LIN {X -205.261,Y 204.855,Z 152.881,A -44.943,B 90.000,C 0.000} C_DIS
LIN {X -207.020,Y 203.080,Z 152.821,A -44.449,B 90.000,C 0.000} C_DIS
LIN {X -207.619,Y 202.471,Z 152.789,A -44.281,B 90.000,C 0.000} C_DIS
LIN {X -208.158,Y 201.917,Z 152.576,A -44.128,B 90.000,C 0.000} C_DIS
LIN {X -208.536,Y 201.526,Z 152.267,A -44.021,B 90.000,C 0.000} C_DIS
LIN {X -208.790,Y 201.263,Z 151.819,A -43.948,B 90.000,C 0.000} C_DIS
LIN {X -208.955,Y 201.092,Z 151.191,A -43.901,B 90.000,C 0.000} C_DIS
LIN {X -209.055,Y 200.988,Z 148.696,A -43.873,B 90.000,C 0.000} C_DIS
LIN {X -209.084,Y 200.957,Z 146.196,A -43.865,B 90.000,C 0.000} C_DIS
LIN {X -209.099,Y 200.942,Z 143.696,A -43.860,B 90.000,C 0.000} C_DIS
LIN {X -209.097,Y 200.943,Z 141.196,A -43.861,B 90.000,C 0.000} C_DIS
LIN {X -209.096,Y 200.945,Z 139.404,A -43.861,B 90.000,C 0.000} C_DIS
LIN {X -208.999,Y 201.046,Z 138.325,A -43.889,B 90.000,C 0.000} C_DIS
LIN {X -208.809,Y 201.244,Z 137.619,A -43.943,B 90.000,C 0.000} C_DIS
LIN {X -208.620,Y 201.439,Z 137.220,A -43.997,B 90.000,C 0.000} C_DIS
LIN {X -208.369,Y 201.699,Z 136.948,A -44.068,B 90.000,C 0.000} C_DIS
LIN {X -208.043,Y 202.035,Z 136.793,A -44.161,B 90.000,C 0.000} C_DIS
LIN {X -207.631,Y 202.458,Z 136.749,A -44.277,B 90.000,C 0.000} C_DIS
LIN {X -206.973,Y 203.130,Z 136.893,A -44.463,B 90.000,C 0.000} C_DIS
LIN {X -205.339,Y 204.778,Z 137.822,A -44.922,B 90.000,C 0.000} C_DIS
LIN {X -203.708,Y 206.402,Z 138.797,A -45.376,B 90.000,C 0.000} C_DIS
LIN {X -202.065,Y 208.014,Z 139.772,A -45.831,B 90.000,C 0.000} C_DIS
LIN {X -200.406,Y 209.610,Z 140.748,A -46.286,B 90.000,C 0.000} C_DIS
LIN {X -198.719,Y 211.200,Z 141.683,A -46.744,B 90.000,C 0.000} C_DIS
LIN {X -197.024,Y 212.788,Z 142.609,A -47.203,B 90.000,C 0.000} C_DIS
LIN {X -195.295,Y 214.371,Z 143.478,A -47.666,B 90.000,C 0.000} C_DIS
LIN {X -193.554,Y 215.952,Z 144.325,A -48.131,B 90.000,C 0.000} C_DIS
LIN {X -191.776,Y 217.532,Z 145.096,A -48.601,B 90.000,C 0.000} C_DIS
LIN {X -189.962,Y 219.119,Z 145.758,A -49.077,B 90.000,C 0.000} C_DIS
LIN {X -189.487,Y 219.532,Z 145.914,A -49.201,B 90.000,C 0.000} C_DIS
LIN {X -188.335,Y 220.522,Z 146.091,A -49.501,B 90.000,C 0.000} C_DIS
LIN {X -187.903,Y 220.890,Z 146.053,A -49.613,B 90.000,C 0.000} C_DIS
LIN {X -187.553,Y 221.188,Z 145.936,A -49.704,B 90.000,C 0.000} C_DIS
LIN {X -187.054,Y 221.609,Z 145.542,A -49.833,B 90.000,C 0.000} C_DIS
LIN {X -186.586,Y 222.004,Z 144.866,A -49.954,B 90.000,C 0.000} C_DIS
LIN {X -186.136,Y 222.381,Z 143.887,A -50.070,B 90.000,C 0.000} C_DIS
LIN {X -185.415,Y 222.982,Z 141.569,A -50.256,B 90.000,C 0.000} C_DIS
LIN {X -184.810,Y 223.484,Z 139.196,A -50.411,B 90.000,C 0.000} C_DIS
LIN {X -184.297,Y 223.908,Z 136.787,A -50.542,B 90.000,C 0.000} C_DIS
LIN {X -183.853,Y 224.272,Z 134.354,A -50.656,B 90.000,C 0.000} C_DIS
LIN {X -183.461,Y 224.593,Z 131.906,A -50.756,B 90.000,C 0.000} C_DIS
LIN {X -183.112,Y 224.878,Z 129.447,A -50.845,B 90.000,C 0.000} C_DIS
LIN {X -182.788,Y 225.141,Z 126.982,A -50.928,B 90.000,C 0.000} C_DIS
LIN {X -182.495,Y 225.379,Z 124.511,A -51.002,B 90.000,C 0.000} C_DIS
LIN {X -182.398,Y 225.457,Z 123.827,A -51.027,B 90.000,C 0.000} C_DIS
LIN {X -182.243,Y 225.583,Z 123.542,A -51.066,B 90.000,C 0.000} C_DIS
LIN {X -181.983,Y 225.792,Z 123.296,A -51.132,B 90.000,C 0.000} C_DIS
LIN {X -181.164,Y 226.450,Z 122.936,A -51.340,B 90.000,C 0.000} C_DIS
LIN {X -180.358,Y 227.093,Z 122.834,A -51.543,B 90.000,C 0.000} C_DIS
LIN {X -179.650,Y 227.653,Z 122.887,A -51.722,B 90.000,C 0.000} C_DIS
LIN {X -179.310,Y 227.921,Z 123.049,A -51.807,B 90.000,C 0.000} C_DIS
LIN {X -179.004,Y 228.162,Z 123.312,A -51.884,B 90.000,C 0.000} C_DIS
LIN {X -178.743,Y 228.366,Z 123.666,A -51.950,B 90.000,C 0.000} C_DIS
LIN {X -178.540,Y 228.525,Z 124.096,A -52.000,B 90.000,C 0.000} C_DIS
LIN {X -178.020,Y 228.930,Z 126.507,A -52.131,B 90.000,C 0.000} C_DIS
LIN {X -177.529,Y 229.310,Z 128.928,A -52.253,B 90.000,C 0.000} C_DIS
LIN {X -177.059,Y 229.673,Z 131.357,A -52.371,B 90.000,C 0.000} C_DIS
LIN {X -176.590,Y 230.035,Z 133.785,A -52.488,B 90.000,C 0.000} C_DIS
LIN {X -176.129,Y 230.386,Z 136.217,A -52.602,B 90.000,C 0.000} C_DIS
LIN {X -175.669,Y 230.737,Z 138.649,A -52.716,B 90.000,C 0.000} C_DIS
LIN {X -175.209,Y 231.087,Z 141.081,A -52.831,B 90.000,C 0.000} C_DIS
LIN {X -174.724,Y 231.455,Z 143.506,A -52.951,B 90.000,C 0.000} C_DIS
LIN {X -174.341,Y 231.744,Z 145.063,A -53.046,B 90.000,C 0.000} C_DIS
LIN {X -174.098,Y 231.926,Z 145.616,A -53.106,B 90.000,C 0.000} C_DIS
LIN {X -173.823,Y 232.133,Z 146.029,A -53.174,B 90.000,C 0.000} C_DIS
LIN {X -173.524,Y 232.357,Z 146.285,A -53.248,B 90.000,C 0.000} C_DIS
LIN {X -172.854,Y 232.855,Z 146.429,A -53.413,B 90.000,C 0.000} C_DIS
LIN {X -171.978,Y 233.503,Z 146.327,A -53.628,B 90.000,C 0.000} C_DIS
LIN {X -170.040,Y 234.913,Z 145.614,A -54.101,B 90.000,C 0.000} C_DIS
LIN {X -168.110,Y 236.292,Z 144.829,A -54.570,B 90.000,C 0.000} C_DIS
LIN {X -166.184,Y 237.651,Z 143.995,A -55.036,B 90.000,C 0.000} C_DIS
LIN {X -164.259,Y 238.992,Z 143.132,A -55.499,B 90.000,C 0.000} C_DIS
LIN {X -162.329,Y 240.307,Z 142.239,A -55.961,B 90.000,C 0.000} C_DIS
LIN {X -160.389,Y 241.607,Z 141.346,A -56.422,B 90.000,C 0.000} C_DIS
LIN {X -158.439,Y 242.891,Z 140.453,A -56.883,B 90.000,C 0.000} C_DIS
LIN {X -156.481,Y 244.158,Z 139.554,A -57.344,B 90.000,C 0.000} C_DIS
LIN {X -154.530,Y 245.397,Z 138.599,A -57.801,B 90.000,C 0.000} C_DIS
LIN {X -152.597,Y 246.605,Z 137.574,A -58.251,B 90.000,C 0.000} C_DIS
LIN {X -151.146,Y 247.497,Z 136.837,A -58.588,B 90.000,C 0.000} C_DIS
LIN {X -150.346,Y 247.984,Z 136.687,A -58.773,B 90.000,C 0.000} C_DIS
LIN {X -149.948,Y 248.225,Z 136.710,A -58.865,B 90.000,C 0.000} C_DIS
LIN {X -149.678,Y 248.388,Z 136.816,A -58.927,B 90.000,C 0.000} C_DIS
LIN {X -149.283,Y 248.625,Z 137.164,A -59.018,B 90.000,C 0.000} C_DIS
LIN {X -148.977,Y 248.809,Z 137.712,A -59.088,B 90.000,C 0.000} C_DIS
LIN {X -148.758,Y 248.940,Z 138.468,A -59.139,B 90.000,C 0.000} C_DIS
LIN {X -148.623,Y 249.021,Z 139.439,A -59.170,B 90.000,C 0.000} C_DIS
LIN {X -148.598,Y 249.036,Z 141.939,A -59.176,B 90.000,C 0.000} C_DIS
LIN {X -148.572,Y 249.051,Z 144.439,A -59.182,B 90.000,C 0.000} C_DIS
LIN {X -148.556,Y 249.060,Z 146.939,A -59.185,B 90.000,C 0.000} C_DIS
LIN {X -148.551,Y 249.063,Z 149.439,A -59.186,B 90.000,C 0.000} C_DIS
LIN {X -148.547,Y 249.066,Z 151.587,A -59.188,B 90.000,C 0.000} C_DIS
LIN {X -147.522,Y 247.348,Z 151.587,A -59.188,B 90.000,C 0.000} C_DIS
WAIT SEC 0.1
RET=EKI_SetBool("oxy","torchState",FALSE)
RET = EKI_Send("oxy","torchState")
LIN {X -138.302,Y 231.889,Z 151.587,A -59.188,B 90.000,C 0.000} C_DIS
LIN {X -139.103,Y 231.409,Z 160.757,A -58.989,B 90.000,C 0.000} C_DIS
LIN {X -148.377,Y 246.837,Z 160.757,A -58.989,B 90.000,C 0.000} C_DIS
LIN {X -149.407,Y 248.551,Z 160.757,A -58.989,B 90.000,C 0.000} C_DIS
WAIT SEC 1
RET=EKI_SetBool("oxy","torchState",TRUE)
RET = EKI_Send("oxy","torchState")
LIN {X -148.004,Y 249.389,Z 160.848,A -59.312,B 90.000,C 0.000} C_DIS
LIN {X -147.671,Y 249.586,Z 163.317,A -59.389,B 90.000,C 0.000} C_DIS
LIN {X -147.269,Y 249.823,Z 165.773,A -59.481,B 90.000,C 0.000} C_DIS
LIN {X -147.069,Y 249.942,Z 166.758,A -59.527,B 90.000,C 0.000} C_DIS
LIN {X -146.655,Y 250.185,Z 168.058,A -59.622,B 90.000,C 0.000} C_DIS
LIN {X -146.177,Y 250.464,Z 168.917,A -59.731,B 90.000,C 0.000} C_DIS
LIN {X -145.706,Y 250.738,Z 169.357,A -59.839,B 90.000,C 0.000} C_DIS
LIN {X -144.278,Y 251.563,Z 169.869,A -60.165,B 90.000,C 0.000} C_DIS
LIN {X -143.823,Y 251.823,Z 170.248,A -60.268,B 90.000,C 0.000} C_DIS
LIN {X -143.521,Y 251.996,Z 170.826,A -60.337,B 90.000,C 0.000} C_DIS
LIN {X -143.469,Y 252.025,Z 171.669,A -60.349,B 90.000,C 0.000} C_DIS
LIN {X -143.814,Y 251.828,Z 174.137,A -60.270,B 90.000,C 0.000} C_DIS
LIN {X -144.166,Y 251.627,Z 176.604,A -60.190,B 90.000,C 0.000} C_DIS
LIN {X -144.676,Y 251.334,Z 179.034,A -60.074,B 90.000,C 0.000} C_DIS
LIN {X -145.317,Y 250.964,Z 181.422,A -59.928,B 90.000,C 0.000} C_DIS
LIN {X -146.090,Y 250.514,Z 183.756,A -59.751,B 90.000,C 0.000} C_DIS
LIN {X -146.998,Y 249.983,Z 186.024,A -59.543,B 90.000,C 0.000} C_DIS
LIN {X -148.038,Y 249.368,Z 188.213,A -59.305,B 90.000,C 0.000} C_DIS
LIN {X -149.207,Y 248.671,Z 190.310,A -59.036,B 90.000,C 0.000} C_DIS
LIN {X -150.499,Y 247.891,Z 192.302,A -58.737,B 90.000,C 0.000} C_DIS
LIN {X -151.923,Y 247.019,Z 194.163,A -58.407,B 90.000,C 0.000} C_DIS
LIN {X -153.430,Y 246.085,Z 195.926,A -58.057,B 90.000,C 0.000} C_DIS
LIN {X -155.015,Y 245.091,Z 197.583,A -57.687,B 90.000,C 0.000} C_DIS
LIN {X -156.684,Y 244.028,Z 199.112,A -57.297,B 90.000,C 0.000} C_DIS
LIN {X -158.440,Y 242.889,Z 200.479,A -56.883,B 90.000,C 0.000} C_DIS
LIN {X -160.220,Y 241.721,Z 201.789,A -56.462,B 90.000,C 0.000} C_DIS
LIN {X -161.274,Y 241.020,Z 202.510,A -56.212,B 90.000,C 0.000} C_DIS
LIN {X -161.782,Y 240.680,Z 202.765,A -56.092,B 90.000,C 0.000} C_DIS
LIN {X -161.983,Y 240.544,Z 202.607,A -56.044,B 90.000,C 0.000} C_DIS
LIN {X -162.981,Y 239.868,Z 200.417,A -55.805,B 90.000,C 0.000} C_DIS
LIN {X -163.955,Y 239.201,Z 198.214,A -55.572,B 90.000,C 0.000} C_DIS
LIN {X -164.908,Y 238.542,Z 195.998,A -55.343,B 90.000,C 0.000} C_DIS
LIN {X -165.861,Y 237.883,Z 193.783,A -55.114,B 90.000,C 0.000} C_DIS
LIN {X -166.809,Y 237.219,Z 191.567,A -54.886,B 90.000,C 0.000} C_DIS
LIN {X -167.752,Y 236.548,Z 189.351,A -54.657,B 90.000,C 0.000} C_DIS
LIN {X -168.695,Y 235.876,Z 187.136,A -54.428,B 90.000,C 0.000} C_DIS
LIN {X -169.638,Y 235.205,Z 184.920,A -54.199,B 90.000,C 0.000} C_DIS
LIN {X -170.568,Y 234.529,Z 182.700,A -53.972,B 90.000,C 0.000} C_DIS
LIN {X -171.491,Y 233.851,Z 180.478,A -53.746,B 90.000,C 0.000} C_DIS
LIN {X -172.415,Y 233.174,Z 178.256,A -53.520,B 90.000,C 0.000} C_DIS
LIN {X -173.333,Y 232.498,Z 176.031,A -53.295,B 90.000,C 0.000} C_DIS
LIN {X -174.194,Y 231.849,Z 173.775,A -53.081,B 90.000,C 0.000} C_DIS
LIN {X -175.056,Y 231.200,Z 171.520,A -52.868,B 90.000,C 0.000} C_DIS
LIN {X -175.920,Y 230.546,Z 169.268,A -52.654,B 90.000,C 0.000} C_DIS
LIN {X -176.795,Y 229.874,Z 167.024,A -52.436,B 90.000,C 0.000} C_DIS
LIN {X -177.679,Y 229.195,Z 164.787,A -52.216,B 90.000,C 0.000} C_DIS
LIN {X -178.719,Y 228.384,Z 162.663,A -51.955,B 90.000,C 0.000} C_DIS
LIN {X -179.553,Y 227.729,Z 161.118,A -51.746,B 90.000,C 0.000} C_DIS
LIN {X -179.641,Y 227.660,Z 160.788,A -51.724,B 90.000,C 0.000} C_DIS
LIN {X -177.672,Y 229.199,Z 160.786,A -52.218,B 90.000,C 0.000} C_DIS
LIN {X -175.689,Y 230.722,Z 160.784,A -52.712,B 90.000,C 0.000} C_DIS
LIN {X -173.694,Y 232.228,Z 160.782,A -53.206,B 90.000,C 0.000} C_DIS
LIN {X -171.685,Y 233.716,Z 160.780,A -53.699,B 90.000,C 0.000} C_DIS
LIN {X -169.664,Y 235.187,Z 160.778,A -54.193,B 90.000,C 0.000} C_DIS
LIN {X -167.630,Y 236.641,Z 160.776,A -54.687,B 90.000,C 0.000} C_DIS
LIN {X -165.583,Y 238.077,Z 160.774,A -55.181,B 90.000,C 0.000} C_DIS
LIN {X -163.525,Y 239.495,Z 160.772,A -55.675,B 90.000,C 0.000} C_DIS
LIN {X -161.454,Y 240.896,Z 160.769,A -56.169,B 90.000,C 0.000} C_DIS
LIN {X -159.371,Y 242.279,Z 160.767,A -56.663,B 90.000,C 0.000} C_DIS
LIN {X -157.277,Y 243.644,Z 160.765,A -57.157,B 90.000,C 0.000} C_DIS
LIN {X -155.171,Y 244.991,Z 160.763,A -57.651,B 90.000,C 0.000} C_DIS
LIN {X -153.053,Y 246.319,Z 160.761,A -58.145,B 90.000,C 0.000} C_DIS
LIN {X -150.924,Y 247.630,Z 160.759,A -58.639,B 90.000,C 0.000} C_DIS
LIN {X -149.407,Y 248.551,Z 160.757,A -58.989,B 90.000,C 0.000} C_DIS
LIN {X -148.377,Y 246.837,Z 160.757,A -58.989,B 90.000,C 0.000} C_DIS
WAIT SEC 0.1
RET=EKI_SetBool("oxy","torchState",FALSE)
RET = EKI_Send("oxy","torchState")
LIN {X -139.103,Y 231.409,Z 160.757,A -58.989,B 90.000,C 0.000} C_DIS
LIN {X -139.074,Y 231.427,Z 126.973,A -58.997,B 90.000,C 0.000} C_DIS
LIN {X -148.346,Y 246.855,Z 126.973,A -58.997,B 90.000,C 0.000} C_DIS
LIN {X -149.376,Y 248.570,Z 126.973,A -58.997,B 90.000,C 0.000} C_DIS
WAIT SEC 1
RET=EKI_SetBool("oxy","torchState",TRUE)
RET = EKI_Send("oxy","torchState")
LIN {X -149.456,Y 248.522,Z 126.964,A -58.978,B 90.000,C 0.000} C_DIS
LIN {X -151.085,Y 247.529,Z 125.348,A -58.601,B 90.000,C 0.000} C_DIS
LIN {X -152.694,Y 246.543,Z 123.709,A -58.228,B 90.000,C 0.000} C_DIS
LIN {X -154.235,Y 245.583,Z 121.990,A -57.870,B 90.000,C 0.000} C_DIS
LIN {X -155.648,Y 244.691,Z 120.131,A -57.540,B 90.000,C 0.000} C_DIS
LIN {X -156.111,Y 244.396,Z 119.238,A -57.431,B 90.000,C 0.000} C_DIS
LIN {X -156.413,Y 244.203,Z 118.302,A -57.360,B 90.000,C 0.000} C_DIS
LIN {X -156.539,Y 244.122,Z 117.113,A -57.331,B 90.000,C 0.000} C_DIS
LIN {X -156.471,Y 244.166,Z 114.614,A -57.347,B 90.000,C 0.000} C_DIS
LIN {X -156.235,Y 244.316,Z 112.130,A -57.402,B 90.000,C 0.000} C_DIS
LIN {X -155.896,Y 244.533,Z 109.663,A -57.482,B 90.000,C 0.000} C_DIS
LIN {X -155.836,Y 244.571,Z 109.402,A -57.496,B 90.000,C 0.000} C_DIS
LIN {X -153.780,Y 245.861,Z 110.003,A -57.975,B 90.000,C 0.000} C_DIS
LIN {X -151.728,Y 247.140,Z 110.635,A -58.453,B 90.000,C 0.000} C_DIS
LIN {X -149.683,Y 248.382,Z 111.361,A -58.925,B 90.000,C 0.000} C_DIS
LIN {X -149.282,Y 248.626,Z 111.504,A -59.018,B 90.000,C 0.000} C_DIS
LIN {X -149.341,Y 248.591,Z 111.613,A -59.005,B 90.000,C 0.000} C_DIS
LIN {X -151.478,Y 247.293,Z 111.578,A -58.511,B 90.000,C 0.000} C_DIS
LIN {X -153.304,Y 246.167,Z 111.730,A -58.087,B 90.000,C 0.000} C_DIS
LIN {X -154.141,Y 245.643,Z 112.053,A -57.892,B 90.000,C 0.000} C_DIS
LIN {X -154.431,Y 245.461,Z 112.286,A -57.824,B 90.000,C 0.000} C_DIS
LIN {X -154.647,Y 245.325,Z 112.591,A -57.774,B 90.000,C 0.000} C_DIS
LIN {X -154.800,Y 245.228,Z 112.983,A -57.738,B 90.000,C 0.000} C_DIS
LIN {X -154.898,Y 245.166,Z 113.481,A -57.715,B 90.000,C 0.000} C_DIS
LIN {X -154.966,Y 245.124,Z 114.860,A -57.699,B 90.000,C 0.000} C_DIS
LIN {X -154.908,Y 245.160,Z 116.152,A -57.713,B 90.000,C 0.000} C_DIS
LIN {X -154.725,Y 245.275,Z 117.383,A -57.755,B 90.000,C 0.000} C_DIS
LIN {X -154.406,Y 245.476,Z 118.611,A -57.830,B 90.000,C 0.000} C_DIS
LIN {X -153.490,Y 246.050,Z 120.865,A -58.043,B 90.000,C 0.000} C_DIS
LIN {X -152.336,Y 246.767,Z 122.963,A -58.312,B 90.000,C 0.000} C_DIS
LIN {X -150.971,Y 247.603,Z 124.883,A -58.628,B 90.000,C 0.000} C_DIS
LIN {X -149.526,Y 248.479,Z 126.726,A -58.962,B 90.000,C 0.000} C_DIS
LIN {X -149.420,Y 248.543,Z 126.863,A -58.986,B 90.000,C 0.000} C_DIS
LIN {X -149.376,Y 248.570,Z 126.973,A -58.997,B 90.000,C 0.000} C_DIS
LIN {X -148.346,Y 246.855,Z 126.973,A -58.997,B 90.000,C 0.000} C_DIS
WAIT SEC 0.1
RET=EKI_SetBool("oxy","torchState",FALSE)
RET = EKI_Send("oxy","torchState")
LIN {X -139.074,Y 231.427,Z 126.973,A -58.997,B 90.000,C 0.000} C_DIS
LIN {X -150.307,Y 224.294,Z 111.089,A -56.173,B 90.000,C 0.000} C_DIS
LIN {X -160.328,Y 239.247,Z 111.089,A -56.173,B 90.000,C 0.000} C_DIS
LIN {X -161.441,Y 240.908,Z 111.089,A -56.173,B 90.000,C 0.000} C_DIS
WAIT SEC 1
RET=EKI_SetBool("oxy","torchState",TRUE)
RET = EKI_Send("oxy","torchState")
LIN {X -163.179,Y 239.733,Z 112.449,A -55.758,B 90.000,C 0.000} C_DIS
LIN {X -164.983,Y 238.492,Z 113.656,A -55.326,B 90.000,C 0.000} C_DIS
LIN {X -166.813,Y 237.213,Z 114.780,A -54.884,B 90.000,C 0.000} C_DIS
LIN {X -168.657,Y 235.905,Z 115.847,A -54.438,B 90.000,C 0.000} C_DIS
LIN {X -170.514,Y 234.565,Z 116.848,A -53.985,B 90.000,C 0.000} C_DIS
LIN {X -172.384,Y 233.195,Z 117.786,A -53.527,B 90.000,C 0.000} C_DIS
LIN {X -174.260,Y 231.802,Z 118.674,A -53.066,B 90.000,C 0.000} C_DIS
LIN {X -176.149,Y 230.369,Z 119.466,A -52.597,B 90.000,C 0.000} C_DIS
LIN {X -178.050,Y 228.903,Z 120.165,A -52.123,B 90.000,C 0.000} C_DIS
LIN {X -178.949,Y 228.204,Z 120.474,A -51.898,B 90.000,C 0.000} C_DIS
LIN {X -180.277,Y 227.157,Z 120.647,A -51.564,B 90.000,C 0.000} C_DIS
LIN {X -181.222,Y 226.403,Z 120.632,A -51.325,B 90.000,C 0.000} C_DIS
LIN {X -182.159,Y 225.651,Z 120.471,A -51.087,B 90.000,C 0.000} C_DIS
LIN {X -184.030,Y 224.125,Z 119.823,A -50.610,B 90.000,C 0.000} C_DIS
LIN {X -185.860,Y 222.607,Z 119.050,A -50.141,B 90.000,C 0.000} C_DIS
LIN {X -187.662,Y 221.092,Z 118.209,A -49.676,B 90.000,C 0.000} C_DIS
LIN {X -189.428,Y 219.582,Z 117.288,A -49.216,B 90.000,C 0.000} C_DIS
LIN {X -191.153,Y 218.078,Z 116.282,A -48.764,B 90.000,C 0.000} C_DIS
LIN {X -192.855,Y 216.574,Z 115.237,A -48.316,B 90.000,C 0.000} C_DIS
LIN {X -194.532,Y 215.070,Z 114.152,A -47.871,B 90.000,C 0.000} C_DIS
LIN {X -196.184,Y 213.566,Z 113.032,A -47.429,B 90.000,C 0.000} C_DIS
LIN {X -197.798,Y 212.074,Z 111.839,A -46.995,B 90.000,C 0.000} C_DIS
LIN {X -199.318,Y 210.647,Z 110.461,A -46.583,B 90.000,C 0.000} C_DIS
LIN {X -200.703,Y 209.325,Z 108.853,A -46.205,B 90.000,C 0.000} C_DIS
LIN {X -202.027,Y 208.048,Z 107.160,A -45.841,B 90.000,C 0.000} C_DIS
LIN {X -203.227,Y 206.878,Z 105.448,A -45.510,B 90.000,C 0.000} C_DIS
LIN {X -203.654,Y 206.458,Z 104.627,A -45.392,B 90.000,C 0.000} C_DIS
LIN {X -203.767,Y 206.346,Z 104.238,A -45.360,B 90.000,C 0.000} C_DIS
LIN {X -203.437,Y 206.672,Z 104.386,A -45.452,B 90.000,C 0.000} C_DIS
LIN {X -201.842,Y 208.224,Z 105.524,A -45.892,B 90.000,C 0.000} C_DIS
LIN {X -200.240,Y 209.770,Z 106.660,A -46.332,B 90.000,C 0.000} C_DIS
LIN {X -198.585,Y 211.326,Z 107.705,A -46.780,B 90.000,C 0.000} C_DIS
LIN {X -196.927,Y 212.882,Z 108.743,A -47.230,B 90.000,C 0.000} C_DIS
LIN {X -195.224,Y 214.440,Z 109.704,A -47.686,B 90.000,C 0.000} C_DIS
LIN {X -193.510,Y 215.990,Z 110.657,A -48.142,B 90.000,C 0.000} C_DIS
LIN {X -191.784,Y 217.527,Z 111.610,A -48.599,B 90.000,C 0.000} C_DIS
LIN {X -190.019,Y 219.068,Z 112.483,A -49.062,B 90.000,C 0.000} C_DIS
LIN {X -188.228,Y 220.609,Z 113.298,A -49.529,B 90.000,C 0.000} C_DIS
LIN {X -186.405,Y 222.150,Z 114.042,A -50.000,B 90.000,C 0.000} C_DIS
LIN {X -184.556,Y 223.693,Z 114.712,A -50.476,B 90.000,C 0.000} C_DIS
LIN {X -182.663,Y 225.243,Z 115.226,A -50.959,B 90.000,C 0.000} C_DIS
LIN {X -182.630,Y 225.269,Z 115.234,A -50.968,B 90.000,C 0.000} C_DIS
LIN {X -180.750,Y 226.781,Z 115.482,A -51.444,B 90.000,C 0.000} C_DIS
LIN {X -178.991,Y 228.172,Z 115.427,A -51.887,B 90.000,C 0.000} C_DIS
LIN {X -177.040,Y 229.686,Z 115.037,A -52.375,B 90.000,C 0.000} C_DIS
LIN {X -175.107,Y 231.163,Z 114.462,A -52.856,B 90.000,C 0.000} C_DIS
LIN {X -173.187,Y 232.604,Z 113.764,A -53.330,B 90.000,C 0.000} C_DIS
LIN {X -171.283,Y 234.009,Z 112.956,A -53.798,B 90.000,C 0.000} C_DIS
LIN {X -169.383,Y 235.388,Z 112.098,A -54.262,B 90.000,C 0.000} C_DIS
LIN {X -167.483,Y 236.744,Z 111.203,A -54.723,B 90.000,C 0.000} C_DIS
LIN {X -165.603,Y 238.066,Z 110.221,A -55.177,B 90.000,C 0.000} C_DIS
LIN {X -163.709,Y 239.370,Z 109.238,A -55.631,B 90.000,C 0.000} C_DIS
LIN {X -161.828,Y 240.641,Z 108.193,A -56.080,B 90.000,C 0.000} C_DIS
LIN {X -159.951,Y 241.900,Z 107.124,A -56.526,B 90.000,C 0.000} C_DIS
LIN {X -158.082,Y 243.120,Z 105.998,A -56.967,B 90.000,C 0.000} C_DIS
LIN {X -156.203,Y 244.337,Z 104.884,A -57.409,B 90.000,C 0.000} C_DIS
LIN {X -156.076,Y 244.418,Z 104.809,A -57.439,B 90.000,C 0.000} C_DIS
LIN {X -155.819,Y 244.582,Z 104.709,A -57.500,B 90.000,C 0.000} C_DIS
LIN {X -155.735,Y 244.635,Z 104.743,A -57.519,B 90.000,C 0.000} C_DIS
LIN {X -156.034,Y 244.445,Z 105.280,A -57.449,B 90.000,C 0.000} C_DIS
LIN {X -157.532,Y 243.480,Z 107.034,A -57.097,B 90.000,C 0.000} C_DIS
LIN {X -159.067,Y 242.480,Z 108.735,A -56.735,B 90.000,C 0.000} C_DIS
LIN {X -160.666,Y 241.423,Z 110.339,A -56.356,B 90.000,C 0.000} C_DIS
LIN {X -161.441,Y 240.908,Z 111.089,A -56.173,B 90.000,C 0.000} C_DIS
LIN {X -160.328,Y 239.247,Z 111.089,A -56.173,B 90.000,C 0.000} C_DIS
WAIT SEC 0.1
RET=EKI_SetBool("oxy","torchState",FALSE)
RET = EKI_Send("oxy","torchState")
LIN {X -150.307,Y 224.294,Z 111.089,A -56.173,B 90.000,C 0.000} C_DIS
LIN {X -152.164,Y 223.038,Z 106.199,A -55.697,B 90.000,C 0.000} C_DIS
LIN {X -162.308,Y 237.908,Z 106.199,A -55.697,B 90.000,C 0.000} C_DIS
LIN {X -163.435,Y 239.560,Z 106.199,A -55.697,B 90.000,C 0.000} C_DIS
WAIT SEC 1
RET=EKI_SetBool("oxy","torchState",TRUE)
RET = EKI_Send("oxy","torchState")
LIN {X -163.575,Y 239.464,Z 106.192,A -55.663,B 90.000,C 0.000} C_DIS
LIN {X -163.681,Y 239.392,Z 106.136,A -55.638,B 90.000,C 0.000} C_DIS
LIN {X -163.820,Y 239.297,Z 105.921,A -55.605,B 90.000,C 0.000} C_DIS
LIN {X -164.813,Y 238.612,Z 103.731,A -55.367,B 90.000,C 0.000} C_DIS
LIN {X -165.781,Y 237.936,Z 101.527,A -55.133,B 90.000,C 0.000} C_DIS
LIN {X -166.748,Y 237.260,Z 99.324,A -54.900,B 90.000,C 0.000} C_DIS
LIN {X -167.714,Y 236.582,Z 97.120,A -54.667,B 90.000,C 0.000} C_DIS
LIN {X -168.674,Y 235.894,Z 94.916,A -54.434,B 90.000,C 0.000} C_DIS
LIN {X -169.634,Y 235.206,Z 92.713,A -54.200,B 90.000,C 0.000} C_DIS
LIN {X -170.593,Y 234.516,Z 90.510,A -53.967,B 90.000,C 0.000} C_DIS
LIN {X -171.553,Y 233.815,Z 88.311,A -53.732,B 90.000,C 0.000} C_DIS
LIN {X -172.450,Y 233.154,Z 86.368,A -53.512,B 90.000,C 0.000} C_DIS
LIN {X -173.673,Y 232.242,Z 84.387,A -53.210,B 90.000,C 0.000} C_DIS
LIN {X -174.914,Y 231.307,Z 82.429,A -52.903,B 90.000,C 0.000} C_DIS
LIN {X -175.617,Y 230.778,Z 81.320,A -52.730,B 90.000,C 0.000} C_DIS
LIN {X -175.703,Y 230.713,Z 80.905,A -52.708,B 90.000,C 0.000} C_DIS
LIN {X -175.604,Y 230.789,Z 80.135,A -52.733,B 90.000,C 0.000} C_DIS
LIN {X -174.968,Y 231.270,Z 77.766,A -52.891,B 90.000,C 0.000} C_DIS
LIN {X -174.142,Y 231.893,Z 75.490,A -53.095,B 90.000,C 0.000} C_DIS
LIN {X -174.024,Y 231.982,Z 75.194,A -53.124,B 90.000,C 0.000} C_DIS
LIN {X -173.228,Y 232.577,Z 73.722,A -53.321,B 90.000,C 0.000} C_DIS
LIN {X -172.272,Y 233.286,Z 72.382,A -53.556,B 90.000,C 0.000} C_DIS
LIN {X -171.261,Y 234.029,Z 71.262,A -53.804,B 90.000,C 0.000} C_DIS
LIN {X -170.170,Y 234.824,Z 70.335,A -54.070,B 90.000,C 0.000} C_DIS
LIN {X -168.953,Y 235.701,Z 69.568,A -54.367,B 90.000,C 0.000} C_DIS
LIN {X -167.565,Y 236.690,Z 68.928,A -54.703,B 90.000,C 0.000} C_DIS
LIN {X -166.410,Y 237.503,Z 68.568,A -54.982,B 90.000,C 0.000} C_DIS
LIN {X -164.358,Y 238.927,Z 68.468,A -55.476,B 90.000,C 0.000} C_DIS
LIN {X -164.146,Y 239.074,Z 68.470,A -55.527,B 90.000,C 0.000} C_DIS
LIN {X -164.072,Y 239.125,Z 68.526,A -55.545,B 90.000,C 0.000} C_DIS
LIN {X -164.188,Y 239.045,Z 68.748,A -55.517,B 90.000,C 0.000} C_DIS
LIN {X -164.530,Y 238.809,Z 69.148,A -55.435,B 90.000,C 0.000} C_DIS
LIN {X -166.385,Y 237.520,Z 70.220,A -54.988,B 90.000,C 0.000} C_DIS
LIN {X -168.178,Y 236.254,Z 71.417,A -54.555,B 90.000,C 0.000} C_DIS
LIN {X -169.310,Y 235.445,Z 72.362,A -54.280,B 90.000,C 0.000} C_DIS
LIN {X -170.408,Y 234.651,Z 73.551,A -54.012,B 90.000,C 0.000} C_DIS
LIN {X -171.502,Y 233.853,Z 75.196,A -53.745,B 90.000,C 0.000} C_DIS
LIN {X -171.887,Y 233.570,Z 76.039,A -53.650,B 90.000,C 0.000} C_DIS
LIN {X -172.172,Y 233.360,Z 76.912,A -53.580,B 90.000,C 0.000} C_DIS
LIN {X -172.418,Y 233.178,Z 78.168,A -53.520,B 90.000,C 0.000} C_DIS
LIN {X -172.458,Y 233.149,Z 79.528,A -53.510,B 90.000,C 0.000} C_DIS
LIN {X -172.301,Y 233.264,Z 81.162,A -53.548,B 90.000,C 0.000} C_DIS
LIN {X -171.868,Y 233.584,Z 82.885,A -53.655,B 90.000,C 0.000} C_DIS
LIN {X -171.047,Y 234.183,Z 85.169,A -53.856,B 90.000,C 0.000} C_DIS
LIN {X -170.227,Y 234.782,Z 87.453,A -54.056,B 90.000,C 0.000} C_DIS
LIN {X -169.376,Y 235.390,Z 89.724,A -54.263,B 90.000,C 0.000} C_DIS
LIN {X -168.518,Y 236.001,Z 91.991,A -54.471,B 90.000,C 0.000} C_DIS
LIN {X -167.659,Y 236.612,Z 94.258,A -54.679,B 90.000,C 0.000} C_DIS
LIN {X -166.801,Y 237.223,Z 96.525,A -54.887,B 90.000,C 0.000} C_DIS
LIN {X -165.941,Y 237.829,Z 98.793,A -55.095,B 90.000,C 0.000} C_DIS
LIN {X -165.079,Y 238.425,Z 101.062,A -55.302,B 90.000,C 0.000} C_DIS
LIN {X -164.216,Y 239.021,Z 103.332,A -55.509,B 90.000,C 0.000} C_DIS
LIN {X -163.353,Y 239.616,Z 105.601,A -55.717,B 90.000,C 0.000} C_DIS
LIN {X -163.328,Y 239.633,Z 105.669,A -55.723,B 90.000,C 0.000} C_DIS
LIN {X -163.291,Y 239.658,Z 105.884,A -55.731,B 90.000,C 0.000} C_DIS
LIN {X -163.352,Y 239.617,Z 106.124,A -55.717,B 90.000,C 0.000} C_DIS
LIN {X -163.435,Y 239.560,Z 106.199,A -55.697,B 90.000,C 0.000} C_DIS
LIN {X -162.308,Y 237.908,Z 106.199,A -55.697,B 90.000,C 0.000} C_DIS
WAIT SEC 0.1
RET=EKI_SetBool("oxy","torchState",FALSE)
RET = EKI_Send("oxy","torchState")
LIN {X -152.164,Y 223.038,Z 106.199,A -55.697,B 90.000,C 0.000} C_DIS
LIN {X -141.870,Y 229.724,Z 103.032,A -58.302,B 90.000,C 0.000} C_DIS
LIN {X -151.328,Y 245.038,Z 103.032,A -58.302,B 90.000,C 0.000} C_DIS
LIN {X -152.379,Y 246.740,Z 103.032,A -58.302,B 90.000,C 0.000} C_DIS
WAIT SEC 1
RET=EKI_SetBool("oxy","torchState",TRUE)
RET = EKI_Send("oxy","torchState")
LIN {X -152.409,Y 246.722,Z 102.859,A -58.295,B 90.000,C 0.000} C_DIS
LIN {X -152.288,Y 246.796,Z 102.521,A -58.323,B 90.000,C 0.000} C_DIS
LIN {X -150.312,Y 248.003,Z 101.580,A -58.780,B 90.000,C 0.000} C_DIS
LIN {X -148.374,Y 249.167,Z 100.511,A -59.227,B 90.000,C 0.000} C_DIS
LIN {X -147.908,Y 249.446,Z 100.241,A -59.334,B 90.000,C 0.000} C_DIS
LIN {X -146.106,Y 250.505,Z 98.870,A -59.747,B 90.000,C 0.000} C_DIS
LIN {X -144.571,Y 251.395,Z 97.332,A -60.098,B 90.000,C 0.000} C_DIS
LIN {X -143.328,Y 252.105,Z 95.636,A -60.381,B 90.000,C 0.000} C_DIS
LIN {X -142.342,Y 252.664,Z 93.741,A -60.605,B 90.000,C 0.000} C_DIS
LIN {X -141.786,Y 252.976,Z 92.230,A -60.731,B 90.000,C 0.000} C_DIS
LIN {X -141.389,Y 253.198,Z 90.624,A -60.820,B 90.000,C 0.000} C_DIS
LIN {X -141.111,Y 253.353,Z 88.144,A -60.883,B 90.000,C 0.000} C_DIS
LIN {X -141.044,Y 253.390,Z 85.900,A -60.898,B 90.000,C 0.000} C_DIS
LIN {X -140.787,Y 253.533,Z 86.205,A -60.957,B 90.000,C 0.000} C_DIS
LIN {X -140.484,Y 253.701,Z 86.731,A -61.025,B 90.000,C 0.000} C_DIS
LIN {X -140.301,Y 253.802,Z 88.839,A -61.066,B 90.000,C 0.000} C_DIS
LIN {X -140.331,Y 253.786,Z 91.236,A -61.060,B 90.000,C 0.000} C_DIS
LIN {X -140.568,Y 253.655,Z 92.829,A -61.006,B 90.000,C 0.000} C_DIS
LIN {X -140.966,Y 253.433,Z 94.320,A -60.916,B 90.000,C 0.000} C_DIS
LIN {X -141.527,Y 253.121,Z 95.713,A -60.789,B 90.000,C 0.000} C_DIS
LIN {X -142.251,Y 252.715,Z 97.010,A -60.625,B 90.000,C 0.000} C_DIS
LIN {X -143.287,Y 252.128,Z 98.343,A -60.390,B 90.000,C 0.000} C_DIS
LIN {X -144.455,Y 251.462,Z 99.548,A -60.124,B 90.000,C 0.000} C_DIS
LIN {X -145.928,Y 250.610,Z 100.652,A -59.788,B 90.000,C 0.000} C_DIS
LIN {X -147.583,Y 249.638,Z 101.587,A -59.409,B 90.000,C 0.000} C_DIS
LIN {X -149.609,Y 248.428,Z 102.411,A -58.943,B 90.000,C 0.000} C_DIS
LIN {X -151.685,Y 247.167,Z 103.004,A -58.463,B 90.000,C 0.000} C_DIS
LIN {X -152.252,Y 246.819,Z 103.103,A -58.331,B 90.000,C 0.000} C_DIS
LIN {X -152.379,Y 246.740,Z 103.032,A -58.302,B 90.000,C 0.000} C_DIS
LIN {X -151.328,Y 245.038,Z 103.032,A -58.302,B 90.000,C 0.000} C_DIS
WAIT SEC 0.1
RET=EKI_SetBool("oxy","torchState",FALSE)
RET = EKI_Send("oxy","torchState")
LIN {X -141.870,Y 229.724,Z 103.032,A -58.302,B 90.000,C 0.000} C_DIS
LIN {X -131.390,Y 235.874,Z 104.704,A -60.881,B 90.000,C 0.000} C_DIS
LIN {X -140.149,Y 251.599,Z 104.704,A -60.881,B 90.000,C 0.000} C_DIS
LIN {X -141.123,Y 253.346,Z 104.704,A -60.881,B 90.000,C 0.000} C_DIS
WAIT SEC 1
RET=EKI_SetBool("oxy","torchState",TRUE)
RET = EKI_Send("oxy","torchState")
LIN {X -139.117,Y 254.450,Z 105.709,A -61.333,B 90.000,C 0.000} C_DIS
LIN {X -138.204,Y 254.950,Z 106.149,A -61.539,B 90.000,C 0.000} C_DIS
LIN {X -136.189,Y 256.032,Z 106.784,A -61.991,B 90.000,C 0.000} C_DIS
LIN {X -135.810,Y 256.234,Z 106.779,A -62.075,B 90.000,C 0.000} C_DIS
LIN {X -135.472,Y 256.412,Z 106.322,A -62.151,B 90.000,C 0.000} C_DIS
LIN {X -134.399,Y 256.975,Z 104.136,A -62.390,B 90.000,C 0.000} C_DIS
LIN {X -133.416,Y 257.488,Z 101.895,A -62.609,B 90.000,C 0.000} C_DIS
LIN {X -132.809,Y 257.802,Z 99.760,A -62.744,B 90.000,C 0.000} C_DIS
LIN {X -132.638,Y 257.890,Z 98.389,A -62.782,B 90.000,C 0.000} C_DIS
LIN {X -134.601,Y 256.866,Z 97.228,A -62.345,B 90.000,C 0.000} C_DIS
LIN {X -136.545,Y 255.843,Z 96.035,A -61.911,B 90.000,C 0.000} C_DIS
LIN {X -137.518,Y 255.319,Z 98.277,A -61.692,B 90.000,C 0.000} C_DIS
LIN {X -138.472,Y 254.804,Z 100.530,A -61.478,B 90.000,C 0.000} C_DIS
LIN {X -139.618,Y 254.178,Z 102.662,A -61.220,B 90.000,C 0.000} C_DIS
LIN {X -140.014,Y 253.961,Z 103.282,A -61.131,B 90.000,C 0.000} C_DIS
LIN {X -141.048,Y 253.388,Z 104.532,A -60.898,B 90.000,C 0.000} C_DIS
LIN {X -141.123,Y 253.346,Z 104.704,A -60.881,B 90.000,C 0.000} C_DIS
LIN {X -140.149,Y 251.599,Z 104.704,A -60.881,B 90.000,C 0.000} C_DIS
WAIT SEC 0.1
RET=EKI_SetBool("oxy","torchState",FALSE)
RET = EKI_Send("oxy","torchState")
LIN {X -131.390,Y 235.874,Z 104.704,A -60.881,B 90.000,C 0.000} C_DIS
LIN {X -124.578,Y 239.542,Z 107.483,A -62.522,B 90.000,C 0.000} C_DIS
LIN {X -132.883,Y 255.511,Z 107.483,A -62.522,B 90.000,C 0.000} C_DIS
LIN {X -133.806,Y 257.286,Z 107.483,A -62.522,B 90.000,C 0.000} C_DIS
WAIT SEC 1
RET=EKI_SetBool("oxy","torchState",TRUE)
RET = EKI_Send("oxy","torchState")
LIN {X -132.836,Y 257.788,Z 105.235,A -62.738,B 90.000,C 0.000} C_DIS
LIN {X -132.043,Y 258.195,Z 102.899,A -62.914,B 90.000,C 0.000} C_DIS
LIN {X -131.462,Y 258.491,Z 100.486,A -63.043,B 90.000,C 0.000} C_DIS
LIN {X -131.165,Y 258.642,Z 98.370,A -63.109,B 90.000,C 0.000} C_DIS
LIN {X -131.194,Y 258.627,Z 95.870,A -63.103,B 90.000,C 0.000} C_DIS
LIN {X -131.290,Y 258.578,Z 94.495,A -63.081,B 90.000,C 0.000} C_DIS
LIN {X -131.688,Y 258.376,Z 92.520,A -62.993,B 90.000,C 0.000} C_DIS
LIN {X -132.314,Y 258.056,Z 90.651,A -62.854,B 90.000,C 0.000} C_DIS
LIN {X -133.194,Y 257.603,Z 88.853,A -62.659,B 90.000,C 0.000} C_DIS
LIN {X -134.306,Y 257.025,Z 87.164,A -62.411,B 90.000,C 0.000} C_DIS
LIN {X -135.864,Y 256.204,Z 85.389,A -62.063,B 90.000,C 0.000} C_DIS
LIN {X -137.578,Y 255.288,Z 83.817,A -61.679,B 90.000,C 0.000} C_DIS
LIN {X -139.395,Y 254.294,Z 82.417,A -61.270,B 90.000,C 0.000} C_DIS
LIN {X -141.223,Y 253.289,Z 81.039,A -60.858,B 90.000,C 0.000} C_DIS
LIN {X -142.847,Y 252.378,Z 79.808,A -60.490,B 90.000,C 0.000} C_DIS
LIN {X -143.257,Y 252.146,Z 79.046,A -60.397,B 90.000,C 0.000} C_DIS
LIN {X -143.083,Y 252.244,Z 79.057,A -60.436,B 90.000,C 0.000} C_DIS
LIN {X -141.199,Y 253.304,Z 79.811,A -60.863,B 90.000,C 0.000} C_DIS
LIN {X -139.222,Y 254.386,Z 80.893,A -61.309,B 90.000,C 0.000} C_DIS
LIN {X -137.262,Y 255.458,Z 81.967,A -61.750,B 90.000,C 0.000} C_DIS
LIN {X -135.518,Y 256.387,Z 83.498,A -62.141,B 90.000,C 0.000} C_DIS
LIN {X -133.866,Y 257.253,Z 85.163,A -62.509,B 90.000,C 0.000} C_DIS
LIN {X -133.271,Y 257.563,Z 85.815,A -62.642,B 90.000,C 0.000} C_DIS
LIN {X -132.193,Y 258.118,Z 87.299,A -62.881,B 90.000,C 0.000} C_DIS
LIN {X -131.331,Y 258.558,Z 88.852,A -63.072,B 90.000,C 0.000} C_DIS
LIN {X -130.682,Y 258.887,Z 90.480,A -63.216,B 90.000,C 0.000} C_DIS
LIN {X -130.036,Y 259.211,Z 92.873,A -63.359,B 90.000,C 0.000} C_DIS
LIN {X -129.670,Y 259.395,Z 94.776,A -63.440,B 90.000,C 0.000} C_DIS
LIN {X -129.587,Y 259.436,Z 97.274,A -63.458,B 90.000,C 0.000} C_DIS
LIN {X -129.673,Y 259.394,Z 99.271,A -63.439,B 90.000,C 0.000} C_DIS
LIN {X -130.023,Y 259.218,Z 101.311,A -63.362,B 90.000,C 0.000} C_DIS
LIN {X -130.550,Y 258.953,Z 103.240,A -63.245,B 90.000,C 0.000} C_DIS
LIN {X -131.476,Y 258.484,Z 105.514,A -63.040,B 90.000,C 0.000} C_DIS
LIN {X -132.625,Y 257.896,Z 107.655,A -62.785,B 90.000,C 0.000} C_DIS
LIN {X -133.052,Y 257.677,Z 108.353,A -62.690,B 90.000,C 0.000} C_DIS
LIN {X -134.452,Y 256.949,Z 110.072,A -62.379,B 90.000,C 0.000} C_DIS
LIN {X -134.918,Y 256.704,Z 109.985,A -62.275,B 90.000,C 0.000} C_DIS
LIN {X -133.925,Y 257.224,Z 107.751,A -62.496,B 90.000,C 0.000} C_DIS
LIN {X -133.806,Y 257.286,Z 107.483,A -62.522,B 90.000,C 0.000} C_DIS
LIN {X -132.883,Y 255.511,Z 107.483,A -62.522,B 90.000,C 0.000} C_DIS
WAIT SEC 0.1
RET=EKI_SetBool("oxy","torchState",FALSE)
RET = EKI_Send("oxy","torchState")
LIN {X -124.578,Y 239.542,Z 107.483,A -62.522,B 90.000,C 0.000} C_DIS
LIN {X -147.605,Y 226.082,Z 82.780,A -56.860,B 90.000,C 0.000} C_DIS
LIN {X -157.445,Y 241.154,Z 82.780,A -56.860,B 90.000,C 0.000} C_DIS
LIN {X -158.538,Y 242.828,Z 82.780,A -56.860,B 90.000,C 0.000} C_DIS
WAIT SEC 1
RET=EKI_SetBool("oxy","torchState",TRUE)
RET = EKI_Send("oxy","torchState")
LIN {X -159.334,Y 242.307,Z 83.710,A -56.672,B 90.000,C 0.000} C_DIS
LIN {X -160.292,Y 241.675,Z 84.484,A -56.446,B 90.000,C 0.000} C_DIS
LIN {X -161.353,Y 240.967,Z 85.049,A -56.193,B 90.000,C 0.000} C_DIS
LIN {X -162.153,Y 240.429,Z 85.292,A -56.003,B 90.000,C 0.000} C_DIS
LIN {X -163.942,Y 239.213,Z 85.458,A -55.576,B 90.000,C 0.000} C_DIS
LIN {X -164.767,Y 238.646,Z 85.365,A -55.378,B 90.000,C 0.000} C_DIS
LIN {X -165.607,Y 238.064,Z 85.121,A -55.176,B 90.000,C 0.000} C_DIS
LIN {X -166.392,Y 237.516,Z 84.749,A -54.987,B 90.000,C 0.000} C_DIS
LIN {X -167.114,Y 237.008,Z 84.259,A -54.812,B 90.000,C 0.000} C_DIS
LIN {X -167.764,Y 236.549,Z 83.660,A -54.655,B 90.000,C 0.000} C_DIS
LIN {X -168.333,Y 236.144,Z 82.963,A -54.517,B 90.000,C 0.000} C_DIS
LIN {X -168.812,Y 235.802,Z 82.177,A -54.401,B 90.000,C 0.000} C_DIS
LIN {X -169.192,Y 235.529,Z 81.313,A -54.308,B 90.000,C 0.000} C_DIS
LIN {X -169.465,Y 235.333,Z 80.379,A -54.242,B 90.000,C 0.000} C_DIS
LIN {X -169.617,Y 235.224,Z 79.076,A -54.205,B 90.000,C 0.000} C_DIS
LIN {X -169.534,Y 235.283,Z 77.767,A -54.225,B 90.000,C 0.000} C_DIS
LIN {X -169.315,Y 235.441,Z 76.834,A -54.279,B 90.000,C 0.000} C_DIS
LIN {X -168.984,Y 235.678,Z 75.969,A -54.359,B 90.000,C 0.000} C_DIS
LIN {X -168.548,Y 235.991,Z 75.178,A -54.465,B 90.000,C 0.000} C_DIS
LIN {X -168.012,Y 236.373,Z 74.468,A -54.595,B 90.000,C 0.000} C_DIS
LIN {X -167.381,Y 236.820,Z 73.845,A -54.748,B 90.000,C 0.000} C_DIS
LIN {X -166.662,Y 237.326,Z 73.318,A -54.922,B 90.000,C 0.000} C_DIS
LIN {X -165.861,Y 237.887,Z 72.893,A -55.115,B 90.000,C 0.000} C_DIS
LIN {X -164.982,Y 238.497,Z 72.578,A -55.326,B 90.000,C 0.000} C_DIS
LIN {X -163.701,Y 239.378,Z 72.436,A -55.633,B 90.000,C 0.000} C_DIS
LIN {X -162.418,Y 240.251,Z 72.504,A -55.940,B 90.000,C 0.000} C_DIS
LIN {X -161.463,Y 240.893,Z 72.794,A -56.167,B 90.000,C 0.000} C_DIS
LIN {X -160.595,Y 241.473,Z 73.220,A -56.374,B 90.000,C 0.000} C_DIS
LIN {X -159.803,Y 241.998,Z 73.788,A -56.561,B 90.000,C 0.000} C_DIS
LIN {X -159.078,Y 242.475,Z 74.504,A -56.733,B 90.000,C 0.000} C_DIS
LIN {X -158.472,Y 242.871,Z 75.294,A -56.876,B 90.000,C 0.000} C_DIS
LIN {X -157.996,Y 243.181,Z 76.134,A -56.988,B 90.000,C 0.000} C_DIS
LIN {X -157.652,Y 243.404,Z 77.015,A -57.069,B 90.000,C 0.000} C_DIS
LIN {X -157.442,Y 243.541,Z 77.929,A -57.119,B 90.000,C 0.000} C_DIS
LIN {X -157.366,Y 243.590,Z 78.868,A -57.136,B 90.000,C 0.000} C_DIS
LIN {X -157.426,Y 243.551,Z 79.823,A -57.122,B 90.000,C 0.000} C_DIS
LIN {X -157.624,Y 243.423,Z 80.786,A -57.076,B 90.000,C 0.000} C_DIS
LIN {X -157.960,Y 243.205,Z 81.749,A -56.996,B 90.000,C 0.000} C_DIS
LIN {X -158.538,Y 242.828,Z 82.780,A -56.860,B 90.000,C 0.000} C_DIS
LIN {X -157.445,Y 241.154,Z 82.780,A -56.860,B 90.000,C 0.000} C_DIS
WAIT SEC 0.1
RET=EKI_SetBool("oxy","torchState",FALSE)
RET = EKI_Send("oxy","torchState")
LIN {X -147.605,Y 226.082,Z 82.780,A -56.860,B 90.000,C 0.000} C_DIS
LIN {X -162.490,Y 215.632,Z 87.325,A -53.000,B 90.000,C 0.000} C_DIS
LIN {X -173.323,Y 230.007,Z 87.325,A -53.000,B 90.000,C 0.000} C_DIS
LIN {X -174.526,Y 231.604,Z 87.325,A -53.000,B 90.000,C 0.000} C_DIS
WAIT SEC 1
RET=EKI_SetBool("oxy","torchState",TRUE)
RET = EKI_Send("oxy","torchState")
LIN {X -174.642,Y 231.517,Z 86.767,A -52.971,B 90.000,C 0.000} C_DIS
LIN {X -174.974,Y 231.266,Z 86.231,A -52.889,B 90.000,C 0.000} C_DIS
LIN {X -175.474,Y 230.887,Z 85.772,A -52.765,B 90.000,C 0.000} C_DIS
LIN {X -176.056,Y 230.444,Z 85.451,A -52.621,B 90.000,C 0.000} C_DIS
LIN {X -176.896,Y 229.799,Z 85.265,A -52.411,B 90.000,C 0.000} C_DIS
LIN {X -177.049,Y 229.682,Z 84.976,A -52.373,B 90.000,C 0.000} C_DIS
LIN {X -177.101,Y 229.641,Z 84.821,A -52.360,B 90.000,C 0.000} C_DIS
LIN {X -179.072,Y 228.103,Z 84.803,A -51.866,B 90.000,C 0.000} C_DIS
LIN {X -181.034,Y 226.554,Z 84.810,A -51.372,B 90.000,C 0.000} C_DIS
LIN {X -182.977,Y 224.981,Z 84.816,A -50.879,B 90.000,C 0.000} C_DIS
LIN {X -183.829,Y 224.292,Z 84.819,A -50.662,B 90.000,C 0.000} C_DIS
LIN {X -183.950,Y 224.193,Z 85.044,A -50.631,B 90.000,C 0.000} C_DIS
LIN {X -184.144,Y 224.033,Z 85.299,A -50.582,B 90.000,C 0.000} C_DIS
LIN {X -185.048,Y 223.287,Z 85.551,A -50.350,B 90.000,C 0.000} C_DIS
LIN {X -185.522,Y 222.894,Z 85.864,A -50.228,B 90.000,C 0.000} C_DIS
LIN {X -185.920,Y 222.562,Z 86.284,A -50.126,B 90.000,C 0.000} C_DIS
LIN {X -186.188,Y 222.338,Z 86.764,A -50.057,B 90.000,C 0.000} C_DIS
LIN {X -186.281,Y 222.260,Z 87.312,A -50.033,B 90.000,C 0.000} C_DIS
LIN {X -186.171,Y 222.352,Z 87.874,A -50.061,B 90.000,C 0.000} C_DIS
LIN {X -185.666,Y 222.774,Z 88.655,A -50.191,B 90.000,C 0.000} C_DIS
LIN {X -184.180,Y 224.003,Z 90.246,A -50.572,B 90.000,C 0.000} C_DIS
LIN {X -183.746,Y 224.360,Z 90.753,A -50.683,B 90.000,C 0.000} C_DIS
LIN {X -181.801,Y 225.930,Z 90.735,A -51.177,B 90.000,C 0.000} C_DIS
LIN {X -179.848,Y 227.491,Z 90.717,A -51.671,B 90.000,C 0.000} C_DIS
LIN {X -177.880,Y 229.032,Z 90.699,A -52.165,B 90.000,C 0.000} C_DIS
LIN {X -177.146,Y 229.607,Z 90.692,A -52.349,B 90.000,C 0.000} C_DIS
LIN {X -176.934,Y 229.771,Z 90.441,A -52.402,B 90.000,C 0.000} C_DIS
LIN {X -175.367,Y 230.968,Z 88.905,A -52.792,B 90.000,C 0.000} C_DIS
LIN {X -175.223,Y 231.077,Z 88.759,A -52.827,B 90.000,C 0.000} C_DIS
LIN {X -174.646,Y 231.514,Z 87.889,A -52.970,B 90.000,C 0.000} C_DIS
LIN {X -174.526,Y 231.604,Z 87.325,A -53.000,B 90.000,C 0.000} C_DIS
LIN {X -173.323,Y 230.007,Z 87.325,A -53.000,B 90.000,C 0.000} C_DIS
WAIT SEC 0.1
RET=EKI_SetBool("oxy","torchState",FALSE)
RET = EKI_Send("oxy","torchState")
LIN {X -162.490,Y 215.632,Z 87.325,A -53.000,B 90.000,C 0.000} C_DIS
LIN {X -172.971,Y 207.319,Z 81.297,A -50.161,B 90.000,C 0.000} C_DIS
LIN {X -184.503,Y 221.140,Z 81.297,A -50.161,B 90.000,C 0.000} C_DIS
LIN {X -185.784,Y 222.675,Z 81.297,A -50.161,B 90.000,C 0.000} C_DIS
WAIT SEC 1
RET=EKI_SetBool("oxy","torchState",TRUE)
RET = EKI_Send("oxy","torchState")
LIN {X -185.727,Y 222.723,Z 80.782,A -50.176,B 90.000,C 0.000} C_DIS
LIN {X -186.269,Y 222.270,Z 78.384,A -50.036,B 90.000,C 0.000} C_DIS
LIN {X -186.485,Y 222.089,Z 77.565,A -49.980,B 90.000,C 0.000} C_DIS
LIN {X -187.253,Y 221.441,Z 75.442,A -49.782,B 90.000,C 0.000} C_DIS
LIN {X -188.185,Y 220.650,Z 73.592,A -49.540,B 90.000,C 0.000} C_DIS
LIN {X -189.281,Y 219.710,Z 72.008,A -49.255,B 90.000,C 0.000} C_DIS
LIN {X -190.542,Y 218.618,Z 70.687,A -48.925,B 90.000,C 0.000} C_DIS
LIN {X -191.491,Y 217.787,Z 69.954,A -48.676,B 90.000,C 0.000} C_DIS
LIN {X -193.227,Y 216.248,Z 69.022,A -48.218,B 90.000,C 0.000} C_DIS
LIN {X -193.647,Y 215.872,Z 68.835,A -48.106,B 90.000,C 0.000} C_DIS
LIN {X -194.710,Y 214.914,Z 68.522,A -47.824,B 90.000,C 0.000} C_DIS
LIN {X -196.472,Y 213.304,Z 68.486,A -47.352,B 90.000,C 0.000} C_DIS
LIN {X -196.420,Y 213.353,Z 68.791,A -47.366,B 90.000,C 0.000} C_DIS
LIN {X -196.249,Y 213.509,Z 69.108,A -47.412,B 90.000,C 0.000} C_DIS
LIN {X -194.572,Y 215.036,Z 70.159,A -47.860,B 90.000,C 0.000} C_DIS
LIN {X -192.940,Y 216.501,Z 71.360,A -48.293,B 90.000,C 0.000} C_DIS
LIN {X -192.307,Y 217.067,Z 71.855,A -48.461,B 90.000,C 0.000} C_DIS
LIN {X -190.839,Y 218.358,Z 73.413,A -48.847,B 90.000,C 0.000} C_DIS
LIN {X -190.661,Y 218.514,Z 73.624,A -48.894,B 90.000,C 0.000} C_DIS
LIN {X -190.027,Y 219.066,Z 74.565,A -49.060,B 90.000,C 0.000} C_DIS
LIN {X -189.521,Y 219.503,Z 75.542,A -49.192,B 90.000,C 0.000} C_DIS
LIN {X -189.144,Y 219.828,Z 76.556,A -49.291,B 90.000,C 0.000} C_DIS
LIN {X -188.897,Y 220.041,Z 77.605,A -49.355,B 90.000,C 0.000} C_DIS
LIN {X -188.780,Y 220.141,Z 78.688,A -49.386,B 90.000,C 0.000} C_DIS
LIN {X -188.794,Y 220.129,Z 79.807,A -49.382,B 90.000,C 0.000} C_DIS
LIN {X -188.916,Y 220.024,Z 80.949,A -49.350,B 90.000,C 0.000} C_DIS
LIN {X -189.484,Y 219.535,Z 83.334,A -49.202,B 90.000,C 0.000} C_DIS
LIN {X -190.258,Y 218.863,Z 85.614,A -48.999,B 90.000,C 0.000} C_DIS
LIN {X -191.035,Y 218.181,Z 87.890,A -48.795,B 90.000,C 0.000} C_DIS
LIN {X -191.812,Y 217.500,Z 90.166,A -48.591,B 90.000,C 0.000} C_DIS
LIN {X -192.587,Y 216.816,Z 92.443,A -48.387,B 90.000,C 0.000} C_DIS
LIN {X -193.357,Y 216.127,Z 94.719,A -48.183,B 90.000,C 0.000} C_DIS
LIN {X -194.126,Y 215.437,Z 96.995,A -47.979,B 90.000,C 0.000} C_DIS
LIN {X -194.895,Y 214.745,Z 99.272,A -47.774,B 90.000,C 0.000} C_DIS
LIN {X -195.657,Y 214.047,Z 101.548,A -47.570,B 90.000,C 0.000} C_DIS
LIN {X -196.418,Y 213.349,Z 103.824,A -47.366,B 90.000,C 0.000} C_DIS
LIN {X -197.129,Y 212.697,Z 105.947,A -47.176,B 90.000,C 0.000} C_DIS
LIN {X -196.978,Y 212.837,Z 106.165,A -47.216,B 90.000,C 0.000} C_DIS
LIN {X -196.803,Y 212.999,Z 106.197,A -47.263,B 90.000,C 0.000} C_DIS
LIN {X -195.919,Y 213.808,Z 104.003,A -47.500,B 90.000,C 0.000} C_DIS
LIN {X -195.034,Y 214.618,Z 101.810,A -47.737,B 90.000,C 0.000} C_DIS
LIN {X -194.150,Y 215.414,Z 99.611,A -47.972,B 90.000,C 0.000} C_DIS
LIN {X -193.268,Y 216.202,Z 97.409,A -48.206,B 90.000,C 0.000} C_DIS
LIN {X -192.385,Y 216.990,Z 95.206,A -48.440,B 90.000,C 0.000} C_DIS
LIN {X -191.502,Y 217.776,Z 93.003,A -48.673,B 90.000,C 0.000} C_DIS
LIN {X -190.616,Y 218.548,Z 90.797,A -48.905,B 90.000,C 0.000} C_DIS
LIN {X -189.729,Y 219.321,Z 88.591,A -49.138,B 90.000,C 0.000} C_DIS
LIN {X -188.844,Y 220.086,Z 86.424,A -49.369,B 90.000,C 0.000} C_DIS
LIN {X -187.689,Y 221.071,Z 84.438,A -49.669,B 90.000,C 0.000} C_DIS
LIN {X -186.483,Y 222.090,Z 82.499,A -49.981,B 90.000,C 0.000} C_DIS
LIN {X -185.784,Y 222.675,Z 81.297,A -50.161,B 90.000,C 0.000} C_DIS
LIN {X -184.503,Y 221.140,Z 81.297,A -50.161,B 90.000,C 0.000} C_DIS
WAIT SEC 0.1
RET=EKI_SetBool("oxy","torchState",FALSE)
RET = EKI_Send("oxy","torchState")
LIN {X -172.971,Y 207.319,Z 81.297,A -50.161,B 90.000,C 0.000} C_DIS
LIN {X -178.370,Y 202.693,Z 80.296,A -48.652,B 90.000,C 0.000} C_DIS
LIN {X -190.261,Y 216.205,Z 80.296,A -48.652,B 90.000,C 0.000} C_DIS
LIN {X -191.582,Y 217.707,Z 80.296,A -48.652,B 90.000,C 0.000} C_DIS
WAIT SEC 1
RET=EKI_SetBool("oxy","torchState",TRUE)
RET = EKI_Send("oxy","torchState")
LIN {X -191.760,Y 217.550,Z 81.091,A -48.605,B 90.000,C 0.000} C_DIS
LIN {X -192.023,Y 217.318,Z 81.839,A -48.536,B 90.000,C 0.000} C_DIS
LIN {X -192.371,Y 217.010,Z 82.543,A -48.444,B 90.000,C 0.000} C_DIS
LIN {X -192.805,Y 216.625,Z 83.205,A -48.330,B 90.000,C 0.000} C_DIS
LIN {X -193.473,Y 216.029,Z 83.962,A -48.153,B 90.000,C 0.000} C_DIS
LIN {X -194.243,Y 215.336,Z 84.587,A -47.948,B 90.000,C 0.000} C_DIS
LIN {X -195.083,Y 214.576,Z 85.059,A -47.724,B 90.000,C 0.000} C_DIS
LIN {X -195.960,Y 213.775,Z 85.356,A -47.489,B 90.000,C 0.000} C_DIS
LIN {X -196.981,Y 212.835,Z 85.448,A -47.215,B 90.000,C 0.000} C_DIS
LIN {X -198.002,Y 211.885,Z 85.364,A -46.940,B 90.000,C 0.000} C_DIS
LIN {X -198.848,Y 211.091,Z 85.096,A -46.711,B 90.000,C 0.000} C_DIS
LIN {X -199.628,Y 210.353,Z 84.679,A -46.499,B 90.000,C 0.000} C_DIS
LIN {X -200.336,Y 209.679,Z 84.119,A -46.305,B 90.000,C 0.000} C_DIS
LIN {X -200.964,Y 209.077,Z 83.421,A -46.133,B 90.000,C 0.000} C_DIS
LIN {X -201.515,Y 208.547,Z 82.578,A -45.982,B 90.000,C 0.000} C_DIS
LIN {X -201.932,Y 208.143,Z 81.604,A -45.868,B 90.000,C 0.000} C_DIS
LIN {X -202.162,Y 207.919,Z 80.826,A -45.804,B 90.000,C 0.000} C_DIS
LIN {X -202.312,Y 207.774,Z 80.032,A -45.763,B 90.000,C 0.000} C_DIS
LIN {X -202.382,Y 207.705,Z 79.232,A -45.744,B 90.000,C 0.000} C_DIS
LIN {X -202.373,Y 207.714,Z 78.436,A -45.746,B 90.000,C 0.000} C_DIS
LIN {X -202.285,Y 207.800,Z 77.651,A -45.771,B 90.000,C 0.000} C_DIS
LIN {X -202.118,Y 207.962,Z 76.886,A -45.816,B 90.000,C 0.000} C_DIS
LIN {X -201.874,Y 208.199,Z 76.151,A -45.884,B 90.000,C 0.000} C_DIS
LIN {X -201.552,Y 208.510,Z 75.455,A -45.972,B 90.000,C 0.000} C_DIS
LIN {X -200.978,Y 209.064,Z 74.574,A -46.130,B 90.000,C 0.000} C_DIS
LIN {X -200.330,Y 209.685,Z 73.831,A -46.307,B 90.000,C 0.000} C_DIS
LIN {X -199.232,Y 210.729,Z 73.037,A -46.606,B 90.000,C 0.000} C_DIS
LIN {X -198.079,Y 211.813,Z 72.565,A -46.919,B 90.000,C 0.000} C_DIS
LIN {X -197.201,Y 212.630,Z 72.455,A -47.156,B 90.000,C 0.000} C_DIS
LIN {X -196.348,Y 213.418,Z 72.473,A -47.385,B 90.000,C 0.000} C_DIS
LIN {X -195.360,Y 214.324,Z 72.723,A -47.650,B 90.000,C 0.000} C_DIS
LIN {X -194.440,Y 215.158,Z 73.172,A -47.896,B 90.000,C 0.000} C_DIS
LIN {X -193.605,Y 215.910,Z 73.813,A -48.118,B 90.000,C 0.000} C_DIS
LIN {X -192.871,Y 216.566,Z 74.635,A -48.312,B 90.000,C 0.000} C_DIS
LIN {X -192.447,Y 216.943,Z 75.269,A -48.424,B 90.000,C 0.000} C_DIS
LIN {X -192.107,Y 217.244,Z 75.932,A -48.514,B 90.000,C 0.000} C_DIS
LIN {X -191.844,Y 217.476,Z 76.638,A -48.583,B 90.000,C 0.000} C_DIS
LIN {X -191.650,Y 217.647,Z 77.406,A -48.634,B 90.000,C 0.000} C_DIS
LIN {X -191.510,Y 217.771,Z 78.871,A -48.671,B 90.000,C 0.000} C_DIS
LIN {X -191.582,Y 217.707,Z 80.296,A -48.652,B 90.000,C 0.000} C_DIS
LIN {X -190.261,Y 216.205,Z 80.296,A -48.652,B 90.000,C 0.000} C_DIS
WAIT SEC 0.1
RET=EKI_SetBool("oxy","torchState",FALSE)
RET = EKI_Send("oxy","torchState")
LIN {X -178.370,Y 202.693,Z 80.296,A -48.652,B 90.000,C 0.000} C_DIS
LIN {X -192.208,Y 189.621,Z 102.586,A -44.612,B 90.000,C 0.000} C_DIS
LIN {X -205.022,Y 202.262,Z 102.586,A -44.612,B 90.000,C 0.000} C_DIS
LIN {X -206.446,Y 203.667,Z 102.586,A -44.612,B 90.000,C 0.000} C_DIS
WAIT SEC 1
RET=EKI_SetBool("oxy","torchState",TRUE)
RET = EKI_Send("oxy","torchState")
LIN {X -208.068,Y 202.008,Z 101.654,A -44.153,B 90.000,C 0.000} C_DIS
LIN {X -209.638,Y 200.378,Z 100.593,A -43.706,B 90.000,C 0.000} C_DIS
LIN {X -211.127,Y 198.809,Z 99.339,A -43.279,B 90.000,C 0.000} C_DIS
LIN {X -212.475,Y 197.368,Z 97.805,A -42.889,B 90.000,C 0.000} C_DIS
LIN {X -213.627,Y 196.120,Z 95.970,A -42.553,B 90.000,C 0.000} C_DIS
LIN {X -214.533,Y 195.130,Z 93.861,A -42.288,B 90.000,C 0.000} C_DIS
LIN {X -215.158,Y 194.440,Z 91.541,A -42.104,B 90.000,C 0.000} C_DIS
LIN {X -215.511,Y 194.049,Z 89.097,A -42.000,B 90.000,C 0.000} C_DIS
LIN {X -215.654,Y 193.890,Z 86.610,A -41.958,B 90.000,C 0.000} C_DIS
LIN {X -215.708,Y 193.830,Z 86.508,A -41.942,B 90.000,C 0.000} C_DIS
LIN {X -215.874,Y 193.645,Z 86.476,A -41.893,B 90.000,C 0.000} C_DIS
LIN {X -215.968,Y 193.540,Z 86.537,A -41.865,B 90.000,C 0.000} C_DIS
LIN {X -216.151,Y 193.336,Z 88.132,A -41.811,B 90.000,C 0.000} C_DIS
LIN {X -216.141,Y 193.347,Z 90.632,A -41.814,B 90.000,C 0.000} C_DIS
LIN {X -216.126,Y 193.364,Z 91.078,A -41.818,B 90.000,C 0.000} C_DIS
LIN {X -215.961,Y 193.548,Z 92.588,A -41.867,B 90.000,C 0.000} C_DIS
LIN {X -215.686,Y 193.855,Z 94.023,A -41.949,B 90.000,C 0.000} C_DIS
LIN {X -215.297,Y 194.286,Z 95.390,A -42.063,B 90.000,C 0.000} C_DIS
LIN {X -214.624,Y 195.029,Z 97.065,A -42.261,B 90.000,C 0.000} C_DIS
LIN {X -213.724,Y 196.015,Z 98.563,A -42.525,B 90.000,C 0.000} C_DIS
LIN {X -212.626,Y 197.205,Z 99.886,A -42.845,B 90.000,C 0.000} C_DIS
LIN {X -211.296,Y 198.630,Z 101.020,A -43.230,B 90.000,C 0.000} C_DIS
LIN {X -209.712,Y 200.302,Z 101.979,A -43.685,B 90.000,C 0.000} C_DIS
LIN {X -208.048,Y 202.028,Z 102.689,A -44.159,B 90.000,C 0.000} C_DIS
LIN {X -206.641,Y 203.469,Z 103.126,A -44.557,B 90.000,C 0.000} C_DIS
LIN {X -206.442,Y 203.670,Z 103.058,A -44.613,B 90.000,C 0.000} C_DIS
LIN {X -206.396,Y 203.717,Z 102.832,A -44.626,B 90.000,C 0.000} C_DIS
LIN {X -206.446,Y 203.667,Z 102.586,A -44.612,B 90.000,C 0.000} C_DIS
LIN {X -205.022,Y 202.262,Z 102.586,A -44.612,B 90.000,C 0.000} C_DIS
WAIT SEC 0.1
RET=EKI_SetBool("oxy","torchState",FALSE)
RET = EKI_Send("oxy","torchState")
LIN {X -192.208,Y 189.621,Z 102.586,A -44.612,B 90.000,C 0.000} C_DIS
LIN {X -192.061,Y 189.770,Z 110.419,A -44.656,B 90.000,C 0.000} C_DIS
LIN {X -204.865,Y 202.421,Z 110.419,A -44.656,B 90.000,C 0.000} C_DIS
LIN {X -206.288,Y 203.827,Z 110.419,A -44.656,B 90.000,C 0.000} C_DIS
WAIT SEC 1
RET=EKI_SetBool("oxy","torchState",TRUE)
RET = EKI_Send("oxy","torchState")
LIN {X -204.575,Y 205.538,Z 109.793,A -45.134,B 90.000,C 0.000} C_DIS
LIN {X -203.653,Y 206.460,Z 109.455,A -45.392,B 90.000,C 0.000} C_DIS
LIN {X -203.605,Y 206.507,Z 109.555,A -45.405,B 90.000,C 0.000} C_DIS
LIN {X -203.297,Y 206.809,Z 112.017,A -45.491,B 90.000,C 0.000} C_DIS
LIN {X -203.083,Y 207.020,Z 114.499,A -45.550,B 90.000,C 0.000} C_DIS
LIN {X -202.999,Y 207.103,Z 116.996,A -45.573,B 90.000,C 0.000} C_DIS
LIN {X -203.038,Y 207.064,Z 118.260,A -45.563,B 90.000,C 0.000} C_DIS
LIN {X -203.274,Y 206.832,Z 119.182,A -45.497,B 90.000,C 0.000} C_DIS
LIN {X -203.591,Y 206.521,Z 119.876,A -45.409,B 90.000,C 0.000} C_DIS
LIN {X -204.784,Y 205.334,Z 121.725,A -45.077,B 90.000,C 0.000} C_DIS
LIN {X -206.023,Y 204.093,Z 123.507,A -44.730,B 90.000,C 0.000} C_DIS
LIN {X -207.322,Y 202.767,Z 125.181,A -44.364,B 90.000,C 0.000} C_DIS
LIN {X -208.634,Y 201.423,Z 126.830,A -43.993,B 90.000,C 0.000} C_DIS
LIN {X -208.786,Y 201.267,Z 127.022,A -43.950,B 90.000,C 0.000} C_DIS
LIN {X -208.872,Y 201.177,Z 127.050,A -43.925,B 90.000,C 0.000} C_DIS
LIN {X -207.737,Y 202.348,Z 125.156,A -44.247,B 90.000,C 0.000} C_DIS
LIN {X -206.618,Y 203.492,Z 123.235,A -44.563,B 90.000,C 0.000} C_DIS
LIN {X -205.648,Y 204.472,Z 121.149,A -44.836,B 90.000,C 0.000} C_DIS
LIN {X -204.874,Y 205.248,Z 118.912,A -45.052,B 90.000,C 0.000} C_DIS
LIN {X -204.574,Y 205.547,Z 117.587,A -45.136,B 90.000,C 0.000} C_DIS
LIN {X -204.402,Y 205.718,Z 116.251,A -45.184,B 90.000,C 0.000} C_DIS
LIN {X -204.348,Y 205.772,Z 114.838,A -45.199,B 90.000,C 0.000} C_DIS
LIN {X -204.394,Y 205.726,Z 113.640,A -45.186,B 90.000,C 0.000} C_DIS
LIN {X -204.573,Y 205.547,Z 112.831,A -45.136,B 90.000,C 0.000} C_DIS
LIN {X -204.744,Y 205.378,Z 112.436,A -45.089,B 90.000,C 0.000} C_DIS
LIN {X -204.966,Y 205.155,Z 112.142,A -45.026,B 90.000,C 0.000} C_DIS
LIN {X -205.268,Y 204.853,Z 111.924,A -44.942,B 90.000,C 0.000} C_DIS
LIN {X -205.676,Y 204.445,Z 111.756,A -44.828,B 90.000,C 0.000} C_DIS
LIN {X -207.428,Y 202.666,Z 111.636,A -44.335,B 90.000,C 0.000} C_DIS
LIN {X -208.788,Y 201.265,Z 111.597,A -43.949,B 90.000,C 0.000} C_DIS
LIN {X -209.012,Y 201.032,Z 111.523,A -43.885,B 90.000,C 0.000} C_DIS
LIN {X -208.888,Y 201.161,Z 111.382,A -43.920,B 90.000,C 0.000} C_DIS
LIN {X -207.198,Y 202.893,Z 110.756,A -44.399,B 90.000,C 0.000} C_DIS
LIN {X -206.288,Y 203.827,Z 110.419,A -44.656,B 90.000,C 0.000} C_DIS
LIN {X -204.865,Y 202.421,Z 110.419,A -44.656,B 90.000,C 0.000} C_DIS
WAIT SEC 0.1
RET=EKI_SetBool("oxy","torchState",FALSE)
RET = EKI_Send("oxy","torchState")
LIN {X -192.061,Y 189.770,Z 110.419,A -44.656,B 90.000,C 0.000} C_DIS
LIN {X -195.807,Y 185.902,Z 111.885,A -43.514,B 90.000,C 0.000} C_DIS
LIN {X -208.861,Y 198.296,Z 111.885,A -43.514,B 90.000,C 0.000} C_DIS
LIN {X -210.311,Y 199.673,Z 111.885,A -43.514,B 90.000,C 0.000} C_DIS
WAIT SEC 1
RET=EKI_SetBool("oxy","torchState",TRUE)
RET = EKI_Send("oxy","torchState")
LIN {X -210.309,Y 199.675,Z 114.384,A -43.514,B 90.000,C 0.000} C_DIS
LIN {X -210.342,Y 199.640,Z 116.884,A -43.505,B 90.000,C 0.000} C_DIS
LIN {X -210.390,Y 199.590,Z 119.383,A -43.491,B 90.000,C 0.000} C_DIS
LIN {X -210.437,Y 199.540,Z 121.882,A -43.478,B 90.000,C 0.000} C_DIS
LIN {X -210.484,Y 199.491,Z 124.381,A -43.464,B 90.000,C 0.000} C_DIS
LIN {X -210.530,Y 199.442,Z 126.880,A -43.451,B 90.000,C 0.000} C_DIS
LIN {X -210.566,Y 199.404,Z 129.379,A -43.440,B 90.000,C 0.000} C_DIS
LIN {X -210.568,Y 199.402,Z 129.681,A -43.440,B 90.000,C 0.000} C_DIS
LIN {X -210.678,Y 199.285,Z 129.954,A -43.408,B 90.000,C 0.000} C_DIS
LIN {X -211.089,Y 198.851,Z 130.570,A -43.290,B 90.000,C 0.000} C_DIS
LIN {X -212.402,Y 197.444,Z 132.165,A -42.910,B 90.000,C 0.000} C_DIS
LIN {X -213.707,Y 196.032,Z 133.763,A -42.530,B 90.000,C 0.000} C_DIS
LIN {X -214.544,Y 195.118,Z 134.844,A -42.285,B 90.000,C 0.000} C_DIS
LIN {X -214.687,Y 194.961,Z 135.351,A -42.243,B 90.000,C 0.000} C_DIS
LIN {X -214.683,Y 194.964,Z 137.851,A -42.244,B 90.000,C 0.000} C_DIS
LIN {X -214.680,Y 194.968,Z 140.351,A -42.245,B 90.000,C 0.000} C_DIS
LIN {X -214.675,Y 194.973,Z 142.851,A -42.247,B 90.000,C 0.000} C_DIS
LIN {X -214.670,Y 194.979,Z 145.351,A -42.248,B 90.000,C 0.000} C_DIS
LIN {X -214.665,Y 194.984,Z 147.851,A -42.249,B 90.000,C 0.000} C_DIS
LIN {X -214.661,Y 194.989,Z 150.351,A -42.251,B 90.000,C 0.000} C_DIS
LIN {X -214.678,Y 194.971,Z 152.851,A -42.246,B 90.000,C 0.000} C_DIS
LIN {X -214.696,Y 194.950,Z 155.350,A -42.240,B 90.000,C 0.000} C_DIS
LIN {X -214.714,Y 194.931,Z 157.706,A -42.235,B 90.000,C 0.000} C_DIS
LIN {X -216.385,Y 193.073,Z 157.771,A -41.741,B 90.000,C 0.000} C_DIS
LIN {X -216.647,Y 192.780,Z 157.770,A -41.664,B 90.000,C 0.000} C_DIS
LIN {X -216.880,Y 192.517,Z 157.671,A -41.594,B 90.000,C 0.000} C_DIS
LIN {X -217.063,Y 192.311,Z 157.329,A -41.540,B 90.000,C 0.000} C_DIS
LIN {X -217.127,Y 192.240,Z 156.669,A -41.521,B 90.000,C 0.000} C_DIS
LIN {X -217.126,Y 192.240,Z 154.169,A -41.521,B 90.000,C 0.000} C_DIS
LIN {X -217.147,Y 192.216,Z 151.670,A -41.515,B 90.000,C 0.000} C_DIS
LIN {X -217.164,Y 192.198,Z 150.156,A -41.510,B 90.000,C 0.000} C_DIS
LIN {X -218.810,Y 190.319,Z 150.057,A -41.016,B 90.000,C 0.000} C_DIS
LIN {X -219.690,Y 189.305,Z 150.003,A -40.751,B 90.000,C 0.000} C_DIS
LIN {X -219.709,Y 189.283,Z 147.503,A -40.746,B 90.000,C 0.000} C_DIS
LIN {X -219.710,Y 189.282,Z 145.003,A -40.745,B 90.000,C 0.000} C_DIS
LIN {X -219.680,Y 189.316,Z 142.504,A -40.754,B 90.000,C 0.000} C_DIS
LIN {X -219.672,Y 189.325,Z 141.817,A -40.756,B 90.000,C 0.000} C_DIS
LIN {X -218.033,Y 191.209,Z 141.701,A -41.250,B 90.000,C 0.000} C_DIS
LIN {X -217.138,Y 192.227,Z 141.640,A -41.518,B 90.000,C 0.000} C_DIS
LIN {X -217.111,Y 192.257,Z 139.140,A -41.526,B 90.000,C 0.000} C_DIS
LIN {X -217.084,Y 192.287,Z 136.640,A -41.534,B 90.000,C 0.000} C_DIS
LIN {X -217.058,Y 192.317,Z 134.141,A -41.541,B 90.000,C 0.000} C_DIS
LIN {X -217.031,Y 192.347,Z 131.641,A -41.549,B 90.000,C 0.000} C_DIS
LIN {X -217.005,Y 192.377,Z 129.142,A -41.557,B 90.000,C 0.000} C_DIS
LIN {X -216.978,Y 192.407,Z 126.642,A -41.565,B 90.000,C 0.000} C_DIS
LIN {X -216.965,Y 192.421,Z 124.142,A -41.569,B 90.000,C 0.000} C_DIS
LIN {X -216.965,Y 192.422,Z 121.642,A -41.569,B 90.000,C 0.000} C_DIS
LIN {X -216.964,Y 192.423,Z 119.142,A -41.569,B 90.000,C 0.000} C_DIS
LIN {X -216.964,Y 192.423,Z 116.643,A -41.569,B 90.000,C 0.000} C_DIS
LIN {X -216.962,Y 192.425,Z 114.143,A -41.570,B 90.000,C 0.000} C_DIS
LIN {X -216.960,Y 192.428,Z 111.643,A -41.571,B 90.000,C 0.000} C_DIS
LIN {X -216.959,Y 192.428,Z 111.421,A -41.571,B 90.000,C 0.000} C_DIS
LIN {X -216.876,Y 192.522,Z 110.649,A -41.596,B 90.000,C 0.000} C_DIS
LIN {X -216.717,Y 192.702,Z 110.386,A -41.643,B 90.000,C 0.000} C_DIS
LIN {X -216.376,Y 193.084,Z 110.318,A -41.744,B 90.000,C 0.000} C_DIS
LIN {X -214.719,Y 194.924,Z 110.663,A -42.233,B 90.000,C 0.000} C_DIS
LIN {X -213.046,Y 196.750,Z 111.003,A -42.723,B 90.000,C 0.000} C_DIS
LIN {X -211.358,Y 198.565,Z 111.328,A -43.212,B 90.000,C 0.000} C_DIS
LIN {X -210.579,Y 199.391,Z 111.531,A -43.437,B 90.000,C 0.000} C_DIS
LIN {X -210.400,Y 199.579,Z 111.680,A -43.488,B 90.000,C 0.000} C_DIS
LIN {X -210.311,Y 199.673,Z 111.885,A -43.514,B 90.000,C 0.000} C_DIS
LIN {X -208.861,Y 198.296,Z 111.885,A -43.514,B 90.000,C 0.000} C_DIS
WAIT SEC 0.1
RET=EKI_SetBool("oxy","torchState",FALSE)
RET = EKI_Send("oxy","torchState")
LIN {X -195.807,Y 185.902,Z 111.885,A -43.514,B 90.000,C 0.000} C_DIS
LIN {X -200.558,Y 180.767,Z 104.719,A -42.029,B 90.000,C 0.000} C_DIS
LIN {X -213.928,Y 192.818,Z 104.719,A -42.029,B 90.000,C 0.000} C_DIS
LIN {X -215.414,Y 194.157,Z 104.719,A -42.029,B 90.000,C 0.000} C_DIS
WAIT SEC 1
RET=EKI_SetBool("oxy","torchState",TRUE)
RET = EKI_Send("oxy","torchState")
LIN {X -215.516,Y 194.044,Z 104.463,A -41.999,B 90.000,C 0.000} C_DIS
LIN {X -216.442,Y 193.010,Z 102.994,A -41.725,B 90.000,C 0.000} C_DIS
LIN {X -217.356,Y 191.979,Z 100.909,A -41.452,B 90.000,C 0.000} C_DIS
LIN {X -218.114,Y 191.118,Z 98.688,A -41.226,B 90.000,C 0.000} C_DIS
LIN {X -218.789,Y 190.345,Z 96.408,A -41.023,B 90.000,C 0.000} C_DIS
LIN {X -218.872,Y 190.250,Z 96.129,A -40.998,B 90.000,C 0.000} C_DIS
LIN {X -218.935,Y 190.177,Z 96.062,A -40.979,B 90.000,C 0.000} C_DIS
LIN {X -219.028,Y 190.071,Z 96.079,A -40.951,B 90.000,C 0.000} C_DIS
LIN {X -220.440,Y 188.426,Z 97.325,A -40.523,B 90.000,C 0.000} C_DIS
LIN {X -221.805,Y 186.822,Z 98.550,A -40.107,B 90.000,C 0.000} C_DIS
LIN {X -221.636,Y 187.022,Z 100.077,A -40.159,B 90.000,C 0.000} C_DIS
LIN {X -221.457,Y 187.235,Z 100.975,A -40.213,B 90.000,C 0.000} C_DIS
LIN {X -220.792,Y 188.018,Z 103.254,A -40.416,B 90.000,C 0.000} C_DIS
LIN {X -220.023,Y 188.917,Z 105.456,A -40.650,B 90.000,C 0.000} C_DIS
LIN {X -219.562,Y 189.453,Z 106.618,A -40.790,B 90.000,C 0.000} C_DIS
LIN {X -219.383,Y 189.661,Z 106.895,A -40.844,B 90.000,C 0.000} C_DIS
LIN {X -218.026,Y 191.219,Z 106.408,A -41.252,B 90.000,C 0.000} C_DIS
LIN {X -216.483,Y 192.964,Z 105.501,A -41.712,B 90.000,C 0.000} C_DIS
LIN {X -215.414,Y 194.157,Z 104.719,A -42.029,B 90.000,C 0.000} C_DIS
LIN {X -213.928,Y 192.818,Z 104.719,A -42.029,B 90.000,C 0.000} C_DIS
WAIT SEC 0.1
RET=EKI_SetBool("oxy","torchState",FALSE)
RET = EKI_Send("oxy","torchState")
LIN {X -200.558,Y 180.767,Z 104.719,A -42.029,B 90.000,C 0.000} C_DIS
LIN {X -205.252,Y 175.418,Z 108.753,A -40.519,B 90.000,C 0.000} C_DIS
LIN {X -218.936,Y 187.113,Z 108.753,A -40.519,B 90.000,C 0.000} C_DIS
LIN {X -220.456,Y 188.412,Z 108.753,A -40.519,B 90.000,C 0.000} C_DIS
WAIT SEC 1
RET=EKI_SetBool("oxy","torchState",TRUE)
RET = EKI_Send("oxy","torchState")
LIN {X -220.148,Y 188.772,Z 109.767,A -40.612,B 90.000,C 0.000} C_DIS
LIN {X -220.164,Y 188.753,Z 109.972,A -40.607,B 90.000,C 0.000} C_DIS
LIN {X -220.284,Y 188.613,Z 110.058,A -40.571,B 90.000,C 0.000} C_DIS
LIN {X -220.454,Y 188.415,Z 110.013,A -40.519,B 90.000,C 0.000} C_DIS
LIN {X -221.528,Y 187.149,Z 108.145,A -40.191,B 90.000,C 0.000} C_DIS
LIN {X -221.873,Y 186.741,Z 107.504,A -40.086,B 90.000,C 0.000} C_DIS
LIN {X -222.710,Y 185.743,Z 105.370,A -39.829,B 90.000,C 0.000} C_DIS
LIN {X -222.720,Y 185.731,Z 105.342,A -39.825,B 90.000,C 0.000} C_DIS
LIN {X -223.341,Y 184.983,Z 103.038,A -39.633,B 90.000,C 0.000} C_DIS
LIN {X -223.361,Y 184.959,Z 102.965,A -39.627,B 90.000,C 0.000} C_DIS
LIN {X -223.772,Y 184.461,Z 100.550,A -39.500,B 90.000,C 0.000} C_DIS
LIN {X -223.806,Y 184.420,Z 100.352,A -39.489,B 90.000,C 0.000} C_DIS
LIN {X -223.999,Y 184.186,Z 97.871,A -39.429,B 90.000,C 0.000} C_DIS
LIN {X -223.982,Y 184.206,Z 95.371,A -39.434,B 90.000,C 0.000} C_DIS
LIN {X -223.701,Y 184.547,Z 92.910,A -39.522,B 90.000,C 0.000} C_DIS
LIN {X -223.253,Y 185.090,Z 90.512,A -39.661,B 90.000,C 0.000} C_DIS
LIN {X -223.176,Y 185.182,Z 90.143,A -39.684,B 90.000,C 0.000} C_DIS
LIN {X -222.720,Y 185.730,Z 88.615,A -39.825,B 90.000,C 0.000} C_DIS
LIN {X -222.134,Y 186.430,Z 87.189,A -40.006,B 90.000,C 0.000} C_DIS
LIN {X -221.405,Y 187.296,Z 85.836,A -40.229,B 90.000,C 0.000} C_DIS
LIN {X -220.208,Y 188.699,Z 84.148,A -40.594,B 90.000,C 0.000} C_DIS
LIN {X -218.939,Y 190.173,Z 82.577,A -40.978,B 90.000,C 0.000} C_DIS
LIN {X -218.849,Y 190.277,Z 82.466,A -41.005,B 90.000,C 0.000} C_DIS
LIN {X -217.422,Y 191.905,Z 81.216,A -41.433,B 90.000,C 0.000} C_DIS
LIN {X -215.901,Y 193.606,Z 80.195,A -41.884,B 90.000,C 0.000} C_DIS
LIN {X -214.360,Y 195.319,Z 79.227,A -42.339,B 90.000,C 0.000} C_DIS
LIN {X -213.980,Y 195.736,Z 79.016,A -42.450,B 90.000,C 0.000} C_DIS
LIN {X -213.986,Y 195.730,Z 79.229,A -42.449,B 90.000,C 0.000} C_DIS
LIN {X -214.080,Y 195.626,Z 79.664,A -42.421,B 90.000,C 0.000} C_DIS
LIN {X -214.248,Y 195.443,Z 79.945,A -42.372,B 90.000,C 0.000} C_DIS
LIN {X -215.675,Y 193.864,Z 81.256,A -41.951,B 90.000,C 0.000} C_DIS
LIN {X -217.076,Y 192.295,Z 82.606,A -41.536,B 90.000,C 0.000} C_DIS
LIN {X -218.420,Y 190.767,Z 84.059,A -41.134,B 90.000,C 0.000} C_DIS
LIN {X -219.674,Y 189.323,Z 85.669,A -40.756,B 90.000,C 0.000} C_DIS
LIN {X -220.792,Y 188.018,Z 87.485,A -40.416,B 90.000,C 0.000} C_DIS
LIN {X -220.916,Y 187.873,Z 87.699,A -40.379,B 90.000,C 0.000} C_DIS
LIN {X -221.638,Y 187.021,Z 89.296,A -40.158,B 90.000,C 0.000} C_DIS
LIN {X -222.187,Y 186.367,Z 90.952,A -39.989,B 90.000,C 0.000} C_DIS
LIN {X -222.569,Y 185.912,Z 92.671,A -39.872,B 90.000,C 0.000} C_DIS
LIN {X -222.785,Y 185.653,Z 94.404,A -39.805,B 90.000,C 0.000} C_DIS
LIN {X -222.872,Y 185.548,Z 96.272,A -39.778,B 90.000,C 0.000} C_DIS
LIN {X -222.782,Y 185.656,Z 98.768,A -39.806,B 90.000,C 0.000} C_DIS
LIN {X -222.660,Y 185.802,Z 100.153,A -39.844,B 90.000,C 0.000} C_DIS
LIN {X -222.242,Y 186.302,Z 102.566,A -39.973,B 90.000,C 0.000} C_DIS
LIN {X -222.157,Y 186.403,Z 103.055,A -39.999,B 90.000,C 0.000} C_DIS
LIN {X -221.560,Y 187.112,Z 105.377,A -40.182,B 90.000,C 0.000} C_DIS
LIN {X -220.837,Y 187.964,Z 107.613,A -40.403,B 90.000,C 0.000} C_DIS
LIN {X -220.456,Y 188.412,Z 108.753,A -40.519,B 90.000,C 0.000} C_DIS
LIN {X -218.936,Y 187.113,Z 108.753,A -40.519,B 90.000,C 0.000} C_DIS
WAIT SEC 0.1
RET=EKI_SetBool("oxy","torchState",FALSE)
RET = EKI_Send("oxy","torchState")
LIN {X -205.252,Y 175.418,Z 108.753,A -40.519,B 90.000,C 0.000} C_DIS
LIN {X -195.170,Y 186.571,Z 160.859,A -43.710,B 90.000,C 0.000} C_DIS
LIN {X -208.181,Y 199.009,Z 160.859,A -43.710,B 90.000,C 0.000} C_DIS
LIN {X -209.627,Y 200.391,Z 160.859,A -43.710,B 90.000,C 0.000} C_DIS
WAIT SEC 1
RET=EKI_SetBool("oxy","torchState",TRUE)
RET = EKI_Send("oxy","torchState")
LIN {X -209.783,Y 200.228,Z 160.941,A -43.665,B 90.000,C 0.000} C_DIS
LIN {X -210.018,Y 199.981,Z 163.417,A -43.598,B 90.000,C 0.000} C_DIS
LIN {X -210.322,Y 199.662,Z 165.878,A -43.511,B 90.000,C 0.000} C_DIS
LIN {X -210.770,Y 199.188,Z 167.985,A -43.382,B 90.000,C 0.000} C_DIS
LIN {X -210.985,Y 198.961,Z 168.594,A -43.320,B 90.000,C 0.000} C_DIS
LIN {X -211.221,Y 198.710,Z 169.057,A -43.252,B 90.000,C 0.000} C_DIS
LIN {X -211.592,Y 198.315,Z 169.478,A -43.145,B 90.000,C 0.000} C_DIS
LIN {X -212.646,Y 197.184,Z 169.885,A -42.839,B 90.000,C 0.000} C_DIS
LIN {X -213.001,Y 196.801,Z 170.274,A -42.736,B 90.000,C 0.000} C_DIS
LIN {X -213.203,Y 196.582,Z 170.867,A -42.677,B 90.000,C 0.000} C_DIS
LIN {X -213.267,Y 196.512,Z 171.692,A -42.659,B 90.000,C 0.000} C_DIS
LIN {X -213.069,Y 196.728,Z 174.174,A -42.717,B 90.000,C 0.000} C_DIS
LIN {X -212.731,Y 197.092,Z 176.624,A -42.815,B 90.000,C 0.000} C_DIS
LIN {X -212.329,Y 197.525,Z 179.053,A -42.931,B 90.000,C 0.000} C_DIS
LIN {X -211.827,Y 198.064,Z 181.442,A -43.077,B 90.000,C 0.000} C_DIS
LIN {X -211.219,Y 198.711,Z 183.779,A -43.252,B 90.000,C 0.000} C_DIS
LIN {X -210.504,Y 199.469,Z 186.052,A -43.458,B 90.000,C 0.000} C_DIS
LIN {X -209.678,Y 200.337,Z 188.246,A -43.695,B 90.000,C 0.000} C_DIS
LIN {X -208.740,Y 201.314,Z 190.347,A -43.962,B 90.000,C 0.000} C_DIS
LIN {X -207.693,Y 202.394,Z 192.344,A -44.260,B 90.000,C 0.000} C_DIS
LIN {X -206.539,Y 203.571,Z 194.223,A -44.585,B 90.000,C 0.000} C_DIS
LIN {X -205.285,Y 204.836,Z 195.977,A -44.937,B 90.000,C 0.000} C_DIS
LIN {X -203.947,Y 206.169,Z 197.615,A -45.310,B 90.000,C 0.000} C_DIS
LIN {X -202.519,Y 207.571,Z 199.114,A -45.706,B 90.000,C 0.000} C_DIS
LIN {X -201.016,Y 209.026,Z 200.482,A -46.119,B 90.000,C 0.000} C_DIS
LIN {X -199.448,Y 210.521,Z 201.730,A -46.547,B 90.000,C 0.000} C_DIS
LIN {X -198.073,Y 211.819,Z 202.726,A -46.921,B 90.000,C 0.000} C_DIS
LIN {X -197.905,Y 211.975,Z 202.722,A -46.966,B 90.000,C 0.000} C_DIS
LIN {X -197.047,Y 212.765,Z 200.511,A -47.196,B 90.000,C 0.000} C_DIS
LIN {X -196.189,Y 213.555,Z 198.300,A -47.427,B 90.000,C 0.000} C_DIS
LIN {X -195.331,Y 214.346,Z 196.089,A -47.657,B 90.000,C 0.000} C_DIS
LIN {X -194.475,Y 215.123,Z 193.872,A -47.886,B 90.000,C 0.000} C_DIS
LIN {X -193.621,Y 215.890,Z 191.652,A -48.113,B 90.000,C 0.000} C_DIS
LIN {X -192.767,Y 216.658,Z 189.431,A -48.340,B 90.000,C 0.000} C_DIS
LIN {X -191.910,Y 217.413,Z 187.207,A -48.565,B 90.000,C 0.000} C_DIS
LIN {X -191.052,Y 218.168,Z 184.984,A -48.791,B 90.000,C 0.000} C_DIS
LIN {X -190.193,Y 218.920,Z 182.760,A -49.017,B 90.000,C 0.000} C_DIS
LIN {X -189.327,Y 219.665,Z 180.536,A -49.242,B 90.000,C 0.000} C_DIS
LIN {X -188.462,Y 220.411,Z 178.313,A -49.468,B 90.000,C 0.000} C_DIS
LIN {X -187.613,Y 221.132,Z 176.075,A -49.688,B 90.000,C 0.000} C_DIS
LIN {X -186.781,Y 221.831,Z 173.823,A -49.903,B 90.000,C 0.000} C_DIS
LIN {X -185.950,Y 222.530,Z 171.572,A -50.117,B 90.000,C 0.000} C_DIS
LIN {X -185.118,Y 223.229,Z 169.320,A -50.332,B 90.000,C 0.000} C_DIS
LIN {X -184.292,Y 223.911,Z 167.061,A -50.544,B 90.000,C 0.000} C_DIS
LIN {X -183.417,Y 224.628,Z 164.832,A -50.767,B 90.000,C 0.000} C_DIS
LIN {X -182.438,Y 225.425,Z 162.674,A -51.016,B 90.000,C 0.000} C_DIS
LIN {X -181.497,Y 226.183,Z 160.972,A -51.255,B 90.000,C 0.000} C_DIS
LIN {X -181.450,Y 226.221,Z 160.776,A -51.267,B 90.000,C 0.000} C_DIS
LIN {X -183.392,Y 224.646,Z 160.760,A -50.773,B 90.000,C 0.000} C_DIS
LIN {X -185.322,Y 223.057,Z 160.760,A -50.279,B 90.000,C 0.000} C_DIS
LIN {X -187.238,Y 221.451,Z 160.764,A -49.785,B 90.000,C 0.000} C_DIS
LIN {X -189.140,Y 219.829,Z 160.768,A -49.291,B 90.000,C 0.000} C_DIS
LIN {X -191.028,Y 218.190,Z 160.772,A -48.797,B 90.000,C 0.000} C_DIS
LIN {X -192.901,Y 216.535,Z 160.776,A -48.304,B 90.000,C 0.000} C_DIS
LIN {X -194.761,Y 214.864,Z 160.780,A -47.810,B 90.000,C 0.000} C_DIS
LIN {X -196.606,Y 213.177,Z 160.784,A -47.316,B 90.000,C 0.000} C_DIS
LIN {X -198.436,Y 211.475,Z 160.789,A -46.822,B 90.000,C 0.000} C_DIS
LIN {X -200.252,Y 209.756,Z 160.793,A -46.328,B 90.000,C 0.000} C_DIS
LIN {X -202.053,Y 208.022,Z 160.797,A -45.834,B 90.000,C 0.000} C_DIS
LIN {X -203.839,Y 206.273,Z 160.801,A -45.340,B 90.000,C 0.000} C_DIS
LIN {X -205.609,Y 204.509,Z 160.805,A -44.846,B 90.000,C 0.000} C_DIS
LIN {X -207.365,Y 202.729,Z 160.809,A -44.352,B 90.000,C 0.000} C_DIS
LIN {X -209.106,Y 200.935,Z 160.822,A -43.858,B 90.000,C 0.000} C_DIS
LIN {X -209.627,Y 200.391,Z 160.859,A -43.710,B 90.000,C 0.000} C_DIS
LIN {X -208.181,Y 199.009,Z 160.859,A -43.710,B 90.000,C 0.000} C_DIS
WAIT SEC 0.1
RET=EKI_SetBool("oxy","torchState",FALSE)
RET = EKI_Send("oxy","torchState")
LIN {X -195.170,Y 186.571,Z 160.859,A -43.710,B 90.000,C 0.000} C_DIS
LIN {X -172.165,Y 207.988,Z 184.815,A -50.383,B 90.000,C 0.000} C_DIS
LIN {X -183.643,Y 221.854,Z 184.815,A -50.383,B 90.000,C 0.000} C_DIS
LIN {X -184.918,Y 223.395,Z 184.815,A -50.383,B 90.000,C 0.000} C_DIS
WAIT SEC 1
RET=EKI_SetBool("oxy","torchState",TRUE)
RET = EKI_Send("oxy","torchState")
LIN {X -184.645,Y 223.621,Z 184.645,A -50.453,B 90.000,C 0.000} C_DIS
LIN {X -182.707,Y 225.197,Z 184.545,A -50.947,B 90.000,C 0.000} C_DIS
LIN {X -180.759,Y 226.765,Z 184.552,A -51.441,B 90.000,C 0.000} C_DIS
LIN {X -178.798,Y 228.315,Z 184.570,A -51.935,B 90.000,C 0.000} C_DIS
LIN {X -176.827,Y 229.852,Z 184.597,A -52.429,B 90.000,C 0.000} C_DIS
LIN {X -176.101,Y 230.409,Z 184.686,A -52.609,B 90.000,C 0.000} C_DIS
LIN {X -175.870,Y 230.585,Z 184.920,A -52.667,B 90.000,C 0.000} C_DIS
LIN {X -175.755,Y 230.673,Z 185.362,A -52.695,B 90.000,C 0.000} C_DIS
LIN {X -175.744,Y 230.682,Z 187.861,A -52.698,B 90.000,C 0.000} C_DIS
LIN {X -175.733,Y 230.690,Z 190.361,A -52.701,B 90.000,C 0.000} C_DIS
LIN {X -175.721,Y 230.699,Z 192.861,A -52.704,B 90.000,C 0.000} C_DIS
LIN {X -175.710,Y 230.708,Z 195.361,A -52.707,B 90.000,C 0.000} C_DIS
LIN {X -175.700,Y 230.716,Z 197.861,A -52.709,B 90.000,C 0.000} C_DIS
LIN {X -175.709,Y 230.708,Z 200.361,A -52.707,B 90.000,C 0.000} C_DIS
LIN {X -175.718,Y 230.701,Z 202.861,A -52.705,B 90.000,C 0.000} C_DIS
LIN {X -175.727,Y 230.694,Z 205.361,A -52.702,B 90.000,C 0.000} C_DIS
LIN {X -175.737,Y 230.687,Z 207.860,A -52.700,B 90.000,C 0.000} C_DIS
LIN {X -175.744,Y 230.682,Z 209.911,A -52.698,B 90.000,C 0.000} C_DIS
LIN {X -175.908,Y 230.557,Z 210.349,A -52.658,B 90.000,C 0.000} C_DIS
LIN {X -176.157,Y 230.366,Z 210.635,A -52.595,B 90.000,C 0.000} C_DIS
LIN {X -176.388,Y 230.189,Z 210.716,A -52.538,B 90.000,C 0.000} C_DIS
LIN {X -177.528,Y 229.311,Z 210.615,A -52.254,B 90.000,C 0.000} C_DIS
LIN {X -177.650,Y 229.217,Z 209.270,A -52.223,B 90.000,C 0.000} C_DIS
LIN {X -177.731,Y 229.155,Z 209.118,A -52.203,B 90.000,C 0.000} C_DIS
LIN {X -177.858,Y 229.055,Z 209.042,A -52.171,B 90.000,C 0.000} C_DIS
LIN {X -179.823,Y 227.510,Z 209.020,A -51.677,B 90.000,C 0.000} C_DIS
LIN {X -181.779,Y 225.953,Z 209.024,A -51.183,B 90.000,C 0.000} C_DIS
LIN {X -182.669,Y 225.238,Z 209.037,A -50.958,B 90.000,C 0.000} C_DIS
LIN {X -183.081,Y 224.903,Z 209.128,A -50.853,B 90.000,C 0.000} C_DIS
LIN {X -183.171,Y 224.830,Z 209.327,A -50.830,B 90.000,C 0.000} C_DIS
LIN {X -183.272,Y 224.747,Z 210.600,A -50.804,B 90.000,C 0.000} C_DIS
LIN {X -184.114,Y 224.058,Z 210.729,A -50.589,B 90.000,C 0.000} C_DIS
LIN {X -184.569,Y 223.683,Z 210.672,A -50.473,B 90.000,C 0.000} C_DIS
LIN {X -184.840,Y 223.460,Z 210.501,A -50.403,B 90.000,C 0.000} C_DIS
LIN {X -184.966,Y 223.355,Z 210.208,A -50.371,B 90.000,C 0.000} C_DIS
LIN {X -185.039,Y 223.295,Z 207.710,A -50.352,B 90.000,C 0.000} C_DIS
LIN {X -185.052,Y 223.284,Z 205.210,A -50.349,B 90.000,C 0.000} C_DIS
LIN {X -185.066,Y 223.273,Z 202.710,A -50.345,B 90.000,C 0.000} C_DIS
LIN {X -185.079,Y 223.262,Z 200.210,A -50.342,B 90.000,C 0.000} C_DIS
LIN {X -185.090,Y 223.252,Z 197.710,A -50.339,B 90.000,C 0.000} C_DIS
LIN {X -185.096,Y 223.247,Z 195.210,A -50.338,B 90.000,C 0.000} C_DIS
LIN {X -185.102,Y 223.242,Z 192.710,A -50.336,B 90.000,C 0.000} C_DIS
LIN {X -185.108,Y 223.237,Z 190.210,A -50.335,B 90.000,C 0.000} C_DIS
LIN {X -185.114,Y 223.232,Z 187.711,A -50.333,B 90.000,C 0.000} C_DIS
LIN {X -185.100,Y 223.244,Z 185.416,A -50.337,B 90.000,C 0.000} C_DIS
LIN {X -185.060,Y 223.278,Z 185.155,A -50.347,B 90.000,C 0.000} C_DIS
LIN {X -184.918,Y 223.395,Z 184.815,A -50.383,B 90.000,C 0.000} C_DIS
LIN {X -183.643,Y 221.854,Z 184.815,A -50.383,B 90.000,C 0.000} C_DIS
WAIT SEC 0.1
RET=EKI_SetBool("oxy","torchState",FALSE)
RET = EKI_Send("oxy","torchState")
LIN {X -172.165,Y 207.988,Z 184.815,A -50.383,B 90.000,C 0.000} C_DIS
LIN {X -262.504,Y 63.181,Z 155.772,A -13.533,B 90.000,C 0.000} C_DIS
LIN {X -280.004,Y 67.393,Z 155.772,A -13.533,B 90.000,C 0.000} C_DIS
LIN {X -281.948,Y 67.861,Z 155.772,A -13.533,B 90.000,C 0.000} C_DIS
WAIT SEC 1
RET=EKI_SetBool("oxy","torchState",TRUE)
RET = EKI_Send("oxy","torchState")
LIN {X -281.936,Y 67.911,Z 155.628,A -13.543,B 90.000,C 0.000} C_DIS
LIN {X -281.927,Y 67.951,Z 154.905,A -13.551,B 90.000,C 0.000} C_DIS
LIN {X -281.902,Y 68.052,Z 154.616,A -13.572,B 90.000,C 0.000} C_DIS
LIN {X -281.893,Y 68.092,Z 153.893,A -13.580,B 90.000,C 0.000} C_DIS
LIN {X -281.869,Y 68.192,Z 153.622,A -13.600,B 90.000,C 0.000} C_DIS
LIN {X -281.859,Y 68.233,Z 153.008,A -13.608,B 90.000,C 0.000} C_DIS
LIN {X -281.834,Y 68.333,Z 152.737,A -13.629,B 90.000,C 0.000} C_DIS
LIN {X -281.825,Y 68.373,Z 152.014,A -13.637,B 90.000,C 0.000} C_DIS
LIN {X -281.800,Y 68.473,Z 151.725,A -13.657,B 90.000,C 0.000} C_DIS
LIN {X -281.791,Y 68.513,Z 151.003,A -13.665,B 90.000,C 0.000} C_DIS
LIN {X -281.766,Y 68.613,Z 150.732,A -13.686,B 90.000,C 0.000} C_DIS
LIN {X -281.756,Y 68.654,Z 150.117,A -13.694,B 90.000,C 0.000} C_DIS
LIN {X -281.744,Y 68.704,Z 149.991,A -13.704,B 90.000,C 0.000} C_DIS
LIN {X -281.732,Y 68.755,Z 149.774,A -13.715,B 90.000,C 0.000} C_DIS
LIN {X -281.732,Y 68.755,Z 148.618,A -13.715,B 90.000,C 0.000} C_DIS
LIN {X -281.757,Y 68.653,Z 148.221,A -13.694,B 90.000,C 0.000} C_DIS
LIN {X -281.766,Y 68.614,Z 147.281,A -13.686,B 90.000,C 0.000} C_DIS
LIN {X -281.791,Y 68.513,Z 146.920,A -13.665,B 90.000,C 0.000} C_DIS
LIN {X -281.800,Y 68.474,Z 145.980,A -13.657,B 90.000,C 0.000} C_DIS
LIN {X -281.825,Y 68.372,Z 145.619,A -13.637,B 90.000,C 0.000} C_DIS
LIN {X -281.834,Y 68.333,Z 144.680,A -13.629,B 90.000,C 0.000} C_DIS
LIN {X -281.859,Y 68.231,Z 144.300,A -13.608,B 90.000,C 0.000} C_DIS
LIN {X -281.868,Y 68.193,Z 143.252,A -13.600,B 90.000,C 0.000} C_DIS
LIN {X -281.893,Y 68.091,Z 142.873,A -13.580,B 90.000,C 0.000} C_DIS
LIN {X -281.902,Y 68.052,Z 141.934,A -13.572,B 90.000,C 0.000} C_DIS
LIN {X -281.927,Y 67.951,Z 141.572,A -13.551,B 90.000,C 0.000} C_DIS
LIN {X -281.936,Y 67.912,Z 140.633,A -13.543,B 90.000,C 0.000} C_DIS
LIN {X -281.961,Y 67.810,Z 140.253,A -13.523,B 90.000,C 0.000} C_DIS
LIN {X -281.970,Y 67.771,Z 139.206,A -13.515,B 90.000,C 0.000} C_DIS
LIN {X -281.994,Y 67.670,Z 138.826,A -13.494,B 90.000,C 0.000} C_DIS
LIN {X -282.004,Y 67.631,Z 137.887,A -13.486,B 90.000,C 0.000} C_DIS
LIN {X -282.028,Y 67.529,Z 137.525,A -13.465,B 90.000,C 0.000} C_DIS
LIN {X -282.037,Y 67.490,Z 136.586,A -13.458,B 90.000,C 0.000} C_DIS
LIN {X -282.062,Y 67.388,Z 136.207,A -13.437,B 90.000,C 0.000} C_DIS
LIN {X -282.071,Y 67.350,Z 135.159,A -13.429,B 90.000,C 0.000} C_DIS
LIN {X -282.095,Y 67.248,Z 134.779,A -13.408,B 90.000,C 0.000} C_DIS
LIN {X -282.105,Y 67.209,Z 133.840,A -13.400,B 90.000,C 0.000} C_DIS
LIN {X -282.129,Y 67.107,Z 133.479,A -13.380,B 90.000,C 0.000} C_DIS
LIN {X -282.138,Y 67.068,Z 132.539,A -13.372,B 90.000,C 0.000} C_DIS
LIN {X -282.162,Y 66.967,Z 132.178,A -13.351,B 90.000,C 0.000} C_DIS
LIN {X -282.171,Y 66.928,Z 131.238,A -13.343,B 90.000,C 0.000} C_DIS
LIN {X -282.196,Y 66.826,Z 130.859,A -13.323,B 90.000,C 0.000} C_DIS
LIN {X -282.205,Y 66.787,Z 129.811,A -13.315,B 90.000,C 0.000} C_DIS
LIN {X -282.229,Y 66.685,Z 129.432,A -13.294,B 90.000,C 0.000} C_DIS
LIN {X -282.238,Y 66.646,Z 128.492,A -13.286,B 90.000,C 0.000} C_DIS
LIN {X -282.262,Y 66.545,Z 128.131,A -13.266,B 90.000,C 0.000} C_DIS
LIN {X -282.271,Y 66.506,Z 127.192,A -13.258,B 90.000,C 0.000} C_DIS
LIN {X -282.295,Y 66.404,Z 126.830,A -13.237,B 90.000,C 0.000} C_DIS
LIN {X -282.304,Y 66.365,Z 125.891,A -13.229,B 90.000,C 0.000} C_DIS
LIN {X -282.328,Y 66.263,Z 125.512,A -13.208,B 90.000,C 0.000} C_DIS
LIN {X -282.337,Y 66.225,Z 124.464,A -13.201,B 90.000,C 0.000} C_DIS
LIN {X -282.361,Y 66.123,Z 124.084,A -13.180,B 90.000,C 0.000} C_DIS
LIN {X -282.370,Y 66.084,Z 123.145,A -13.172,B 90.000,C 0.000} C_DIS
LIN {X -282.394,Y 65.982,Z 122.784,A -13.151,B 90.000,C 0.000} C_DIS
LIN {X -282.403,Y 65.943,Z 121.844,A -13.143,B 90.000,C 0.000} C_DIS
LIN {X -282.427,Y 65.841,Z 121.483,A -13.123,B 90.000,C 0.000} C_DIS
LIN {X -282.436,Y 65.802,Z 120.543,A -13.115,B 90.000,C 0.000} C_DIS
LIN {X -282.460,Y 65.700,Z 120.164,A -13.094,B 90.000,C 0.000} C_DIS
LIN {X -282.469,Y 65.662,Z 119.116,A -13.086,B 90.000,C 0.000} C_DIS
LIN {X -282.492,Y 65.560,Z 118.737,A -13.066,B 90.000,C 0.000} C_DIS
LIN {X -282.501,Y 65.521,Z 117.797,A -13.058,B 90.000,C 0.000} C_DIS
LIN {X -282.525,Y 65.419,Z 117.418,A -13.037,B 90.000,C 0.000} C_DIS
LIN {X -282.534,Y 65.380,Z 116.370,A -13.029,B 90.000,C 0.000} C_DIS
LIN {X -282.558,Y 65.278,Z 115.991,A -13.009,B 90.000,C 0.000} C_DIS
LIN {X -282.567,Y 65.239,Z 115.051,A -13.001,B 90.000,C 0.000} C_DIS
LIN {X -282.590,Y 65.137,Z 114.690,A -12.980,B 90.000,C 0.000} C_DIS
LIN {X -282.599,Y 65.098,Z 113.751,A -12.972,B 90.000,C 0.000} C_DIS
LIN {X -282.622,Y 64.996,Z 113.389,A -12.951,B 90.000,C 0.000} C_DIS
LIN {X -282.631,Y 64.957,Z 112.450,A -12.944,B 90.000,C 0.000} C_DIS
LIN {X -282.655,Y 64.855,Z 112.070,A -12.923,B 90.000,C 0.000} C_DIS
LIN {X -282.664,Y 64.817,Z 111.023,A -12.915,B 90.000,C 0.000} C_DIS
LIN {X -282.687,Y 64.715,Z 110.643,A -12.894,B 90.000,C 0.000} C_DIS
LIN {X -282.696,Y 64.676,Z 109.704,A -12.886,B 90.000,C 0.000} C_DIS
LIN {X -282.719,Y 64.574,Z 109.342,A -12.866,B 90.000,C 0.000} C_DIS
LIN {X -282.728,Y 64.535,Z 108.403,A -12.858,B 90.000,C 0.000} C_DIS
LIN {X -282.752,Y 64.433,Z 108.024,A -12.837,B 90.000,C 0.000} C_DIS
LIN {X -282.760,Y 64.394,Z 106.976,A -12.829,B 90.000,C 0.000} C_DIS
LIN {X -282.784,Y 64.292,Z 106.596,A -12.809,B 90.000,C 0.000} C_DIS
LIN {X -282.792,Y 64.253,Z 105.657,A -12.801,B 90.000,C 0.000} C_DIS
LIN {X -282.816,Y 64.151,Z 105.296,A -12.780,B 90.000,C 0.000} C_DIS
LIN {X -282.824,Y 64.112,Z 104.356,A -12.772,B 90.000,C 0.000} C_DIS
LIN {X -282.848,Y 64.010,Z 103.995,A -12.752,B 90.000,C 0.000} C_DIS
LIN {X -282.856,Y 63.971,Z 103.055,A -12.744,B 90.000,C 0.000} C_DIS
LIN {X -282.879,Y 63.869,Z 102.676,A -12.723,B 90.000,C 0.000} C_DIS
LIN {X -282.888,Y 63.830,Z 101.628,A -12.715,B 90.000,C 0.000} C_DIS
LIN {X -282.911,Y 63.728,Z 101.249,A -12.694,B 90.000,C 0.000} C_DIS
LIN {X -282.920,Y 63.689,Z 100.309,A -12.687,B 90.000,C 0.000} C_DIS
LIN {X -282.943,Y 63.587,Z 99.948,A -12.666,B 90.000,C 0.000} C_DIS
LIN {X -282.952,Y 63.548,Z 99.009,A -12.658,B 90.000,C 0.000} C_DIS
LIN {X -282.975,Y 63.446,Z 98.629,A -12.637,B 90.000,C 0.000} C_DIS
LIN {X -282.983,Y 63.407,Z 97.581,A -12.629,B 90.000,C 0.000} C_DIS
LIN {X -283.006,Y 63.305,Z 97.202,A -12.609,B 90.000,C 0.000} C_DIS
LIN {X -283.015,Y 63.266,Z 96.263,A -12.601,B 90.000,C 0.000} C_DIS
LIN {X -283.038,Y 63.164,Z 95.901,A -12.580,B 90.000,C 0.000} C_DIS
LIN {X -283.046,Y 63.125,Z 94.962,A -12.572,B 90.000,C 0.000} C_DIS
LIN {X -283.069,Y 63.023,Z 94.601,A -12.552,B 90.000,C 0.000} C_DIS
LIN {X -283.078,Y 62.984,Z 93.661,A -12.544,B 90.000,C 0.000} C_DIS
LIN {X -283.100,Y 62.882,Z 93.300,A -12.523,B 90.000,C 0.000} C_DIS
LIN {X -283.109,Y 62.843,Z 92.360,A -12.515,B 90.000,C 0.000} C_DIS
LIN {X -283.132,Y 62.741,Z 91.981,A -12.495,B 90.000,C 0.000} C_DIS
LIN {X -283.140,Y 62.702,Z 90.933,A -12.487,B 90.000,C 0.000} C_DIS
LIN {X -283.163,Y 62.600,Z 90.554,A -12.466,B 90.000,C 0.000} C_DIS
LIN {X -283.172,Y 62.560,Z 89.614,A -12.458,B 90.000,C 0.000} C_DIS
LIN {X -283.194,Y 62.458,Z 89.253,A -12.437,B 90.000,C 0.000} C_DIS
LIN {X -283.203,Y 62.419,Z 88.314,A -12.430,B 90.000,C 0.000} C_DIS
LIN {X -283.225,Y 62.317,Z 87.934,A -12.409,B 90.000,C 0.000} C_DIS
LIN {X -283.234,Y 62.278,Z 86.886,A -12.401,B 90.000,C 0.000} C_DIS
LIN {X -283.256,Y 62.176,Z 86.507,A -12.380,B 90.000,C 0.000} C_DIS
LIN {X -283.265,Y 62.137,Z 85.568,A -12.372,B 90.000,C 0.000} C_DIS
LIN {X -283.287,Y 62.035,Z 85.206,A -12.352,B 90.000,C 0.000} C_DIS
LIN {X -283.296,Y 61.996,Z 84.267,A -12.344,B 90.000,C 0.000} C_DIS
LIN {X -283.318,Y 61.894,Z 83.887,A -12.323,B 90.000,C 0.000} C_DIS
LIN {X -283.327,Y 61.855,Z 82.840,A -12.315,B 90.000,C 0.000} C_DIS
LIN {X -283.349,Y 61.753,Z 82.460,A -12.295,B 90.000,C 0.000} C_DIS
LIN {X -283.357,Y 61.713,Z 81.521,A -12.287,B 90.000,C 0.000} C_DIS
LIN {X -283.380,Y 61.611,Z 81.159,A -12.266,B 90.000,C 0.000} C_DIS
LIN {X -283.388,Y 61.572,Z 80.220,A -12.258,B 90.000,C 0.000} C_DIS
LIN {X -283.410,Y 61.470,Z 79.859,A -12.238,B 90.000,C 0.000} C_DIS
LIN {X -283.419,Y 61.431,Z 78.919,A -12.230,B 90.000,C 0.000} C_DIS
LIN {X -283.441,Y 61.329,Z 78.558,A -12.209,B 90.000,C 0.000} C_DIS
LIN {X -283.449,Y 61.290,Z 77.618,A -12.201,B 90.000,C 0.000} C_DIS
LIN {X -283.472,Y 61.187,Z 77.239,A -12.180,B 90.000,C 0.000} C_DIS
LIN {X -283.480,Y 61.149,Z 76.191,A -12.173,B 90.000,C 0.000} C_DIS
LIN {X -283.502,Y 61.046,Z 75.812,A -12.152,B 90.000,C 0.000} C_DIS
LIN {X -283.510,Y 61.007,Z 74.872,A -12.144,B 90.000,C 0.000} C_DIS
LIN {X -283.532,Y 60.905,Z 74.493,A -12.123,B 90.000,C 0.000} C_DIS
LIN {X -283.541,Y 60.866,Z 73.445,A -12.115,B 90.000,C 0.000} C_DIS
LIN {X -283.563,Y 60.764,Z 73.066,A -12.095,B 90.000,C 0.000} C_DIS
LIN {X -283.571,Y 60.724,Z 72.126,A -12.087,B 90.000,C 0.000} C_DIS
LIN {X -283.593,Y 60.622,Z 71.765,A -12.066,B 90.000,C 0.000} C_DIS
LIN {X -283.601,Y 60.583,Z 70.826,A -12.058,B 90.000,C 0.000} C_DIS
LIN {X -283.623,Y 60.481,Z 70.464,A -12.038,B 90.000,C 0.000} C_DIS
LIN {X -283.631,Y 60.442,Z 69.525,A -12.030,B 90.000,C 0.000} C_DIS
LIN {X -283.653,Y 60.340,Z 69.145,A -12.009,B 90.000,C 0.000} C_DIS
LIN {X -283.661,Y 60.301,Z 68.098,A -12.001,B 90.000,C 0.000} C_DIS
LIN {X -283.683,Y 60.198,Z 67.718,A -11.981,B 90.000,C 0.000} C_DIS
LIN {X -283.692,Y 60.159,Z 66.779,A -11.973,B 90.000,C 0.000} C_DIS
LIN {X -283.713,Y 60.058,Z 66.462,A -11.952,B 90.000,C 0.000} C_DIS
LIN {X -283.725,Y 60.002,Z 65.690,A -11.941,B 90.000,C 0.000} C_DIS
LIN {X -283.766,Y 59.808,Z 65.409,A -11.902,B 90.000,C 0.000} C_DIS
LIN {X -283.766,Y 59.808,Z 65.409,A -11.902,B 90.000,C 0.000} C_DIS
LIN {X -283.817,Y 59.564,Z 65.209,A -11.852,B 90.000,C 0.000} C_DIS
LIN {X -283.878,Y 59.275,Z 65.158,A -11.794,B 90.000,C 0.000} C_DIS
LIN {X -283.939,Y 58.982,Z 65.200,A -11.735,B 90.000,C 0.000} C_DIS
LIN {X -283.992,Y 58.726,Z 65.404,A -11.683,B 90.000,C 0.000} C_DIS
LIN {X -284.313,Y 57.149,Z 67.317,A -11.365,B 90.000,C 0.000} C_DIS
LIN {X -284.629,Y 55.554,Z 69.215,A -11.044,B 90.000,C 0.000} C_DIS
LIN {X -284.934,Y 53.968,Z 71.123,A -10.725,B 90.000,C 0.000} C_DIS
LIN {X -285.232,Y 52.368,Z 73.021,A -10.404,B 90.000,C 0.000} C_DIS
LIN {X -285.522,Y 50.767,Z 74.919,A -10.082,B 90.000,C 0.000} C_DIS
LIN {X -285.802,Y 49.165,Z 76.817,A -9.761,B 90.000,C 0.000} C_DIS
LIN {X -286.072,Y 47.570,Z 78.724,A -9.441,B 90.000,C 0.000} C_DIS
LIN {X -286.334,Y 45.966,Z 80.623,A -9.120,B 90.000,C 0.000} C_DIS
LIN {X -286.587,Y 44.360,Z 82.521,A -8.799,B 90.000,C 0.000} C_DIS
LIN {X -286.831,Y 42.751,Z 84.420,A -8.477,B 90.000,C 0.000} C_DIS
LIN {X -287.065,Y 41.153,Z 86.328,A -8.158,B 90.000,C 0.000} C_DIS
LIN {X -287.291,Y 39.542,Z 88.226,A -7.837,B 90.000,C 0.000} C_DIS
LIN {X -287.509,Y 37.930,Z 90.124,A -7.515,B 90.000,C 0.000} C_DIS
LIN {X -287.717,Y 36.316,Z 92.022,A -7.194,B 90.000,C 0.000} C_DIS
LIN {X -287.915,Y 34.713,Z 93.930,A -6.875,B 90.000,C 0.000} C_DIS
LIN {X -288.105,Y 33.098,Z 95.828,A -6.553,B 90.000,C 0.000} C_DIS
LIN {X -288.286,Y 31.481,Z 97.726,A -6.232,B 90.000,C 0.000} C_DIS
LIN {X -288.457,Y 29.875,Z 99.634,A -5.913,B 90.000,C 0.000} C_DIS
LIN {X -288.599,Y 28.471,Z 101.253,A -5.634,B 90.000,C 0.000} C_DIS
LIN {X -288.626,Y 28.200,Z 101.646,A -5.580,B 90.000,C 0.000} C_DIS
LIN {X -288.636,Y 28.099,Z 101.758,A -5.560,B 90.000,C 0.000} C_DIS
LIN {X -288.640,Y 28.056,Z 101.879,A -5.552,B 90.000,C 0.000} C_DIS
LIN {X -288.642,Y 28.035,Z 101.970,A -5.548,B 90.000,C 0.000} C_DIS
LIN {X -288.647,Y 27.984,Z 102.008,A -5.538,B 90.000,C 0.000} C_DIS
LIN {X -288.652,Y 27.931,Z 102.423,A -5.527,B 90.000,C 0.000} C_DIS
LIN {X -288.655,Y 27.894,Z 104.923,A -5.520,B 90.000,C 0.000} C_DIS
LIN {X -288.655,Y 27.893,Z 104.971,A -5.519,B 90.000,C 0.000} C_DIS
LIN {X -288.660,Y 27.850,Z 105.156,A -5.511,B 90.000,C 0.000} C_DIS
LIN {X -288.667,Y 27.769,Z 105.187,A -5.495,B 90.000,C 0.000} C_DIS
LIN {X -288.677,Y 27.667,Z 105.209,A -5.475,B 90.000,C 0.000} C_DIS
LIN {X -288.681,Y 27.625,Z 105.260,A -5.466,B 90.000,C 0.000} C_DIS
LIN {X -288.687,Y 27.561,Z 105.311,A -5.454,B 90.000,C 0.000} C_DIS
LIN {X -288.716,Y 27.257,Z 105.353,A -5.393,B 90.000,C 0.000} C_DIS
LIN {X -288.722,Y 27.193,Z 105.404,A -5.381,B 90.000,C 0.000} C_DIS
LIN {X -288.725,Y 27.160,Z 105.455,A -5.374,B 90.000,C 0.000} C_DIS
LIN {X -288.733,Y 27.082,Z 105.476,A -5.358,B 90.000,C 0.000} C_DIS
LIN {X -288.745,Y 26.950,Z 105.529,A -5.332,B 90.000,C 0.000} C_DIS
LIN {X -288.759,Y 26.797,Z 105.654,A -5.302,B 90.000,C 0.000} C_DIS
LIN {X -288.771,Y 26.670,Z 105.806,A -5.277,B 90.000,C 0.000} C_DIS
LIN {X -288.776,Y 26.618,Z 105.937,A -5.266,B 90.000,C 0.000} C_DIS
LIN {X -288.784,Y 26.528,Z 106.085,A -5.248,B 90.000,C 0.000} C_DIS
LIN {X -288.789,Y 26.474,Z 106.127,A -5.238,B 90.000,C 0.000} C_DIS
LIN {X -288.784,Y 26.528,Z 106.169,A -5.248,B 90.000,C 0.000} C_DIS
LIN {X -288.778,Y 26.593,Z 106.297,A -5.261,B 90.000,C 0.000} C_DIS
LIN {X -288.774,Y 26.639,Z 106.817,A -5.270,B 90.000,C 0.000} C_DIS
LIN {X -288.765,Y 26.740,Z 107.007,A -5.291,B 90.000,C 0.000} C_DIS
LIN {X -288.761,Y 26.783,Z 107.415,A -5.299,B 90.000,C 0.000} C_DIS
LIN {X -288.751,Y 26.884,Z 107.585,A -5.319,B 90.000,C 0.000} C_DIS
LIN {X -288.747,Y 26.926,Z 107.993,A -5.328,B 90.000,C 0.000} C_DIS
LIN {X -288.738,Y 27.028,Z 108.163,A -5.348,B 90.000,C 0.000} C_DIS
LIN {X -288.734,Y 27.070,Z 108.571,A -5.356,B 90.000,C 0.000} C_DIS
LIN {X -288.724,Y 27.172,Z 108.741,A -5.376,B 90.000,C 0.000} C_DIS
LIN {X -288.720,Y 27.214,Z 109.149,A -5.385,B 90.000,C 0.000} C_DIS
LIN {X -288.711,Y 27.316,Z 109.319,A -5.405,B 90.000,C 0.000} C_DIS
LIN {X -288.707,Y 27.358,Z 109.727,A -5.413,B 90.000,C 0.000} C_DIS
LIN {X -288.697,Y 27.460,Z 109.897,A -5.433,B 90.000,C 0.000} C_DIS
LIN {X -288.693,Y 27.502,Z 110.305,A -5.442,B 90.000,C 0.000} C_DIS
LIN {X -288.683,Y 27.604,Z 110.475,A -5.462,B 90.000,C 0.000} C_DIS
LIN {X -288.679,Y 27.646,Z 110.884,A -5.470,B 90.000,C 0.000} C_DIS
LIN {X -288.674,Y 27.697,Z 110.968,A -5.480,B 90.000,C 0.000} C_DIS
LIN {X -288.669,Y 27.750,Z 111.348,A -5.491,B 90.000,C 0.000} C_DIS
LIN {X -288.669,Y 27.750,Z 113.480,A -5.491,B 90.000,C 0.000} C_DIS
LIN {X -288.680,Y 27.634,Z 115.977,A -5.468,B 90.000,C 0.000} C_DIS
LIN {X -288.682,Y 27.615,Z 118.477,A -5.464,B 90.000,C 0.000} C_DIS
LIN {X -288.691,Y 27.523,Z 120.975,A -5.446,B 90.000,C 0.000} C_DIS
LIN {X -288.695,Y 27.484,Z 123.475,A -5.438,B 90.000,C 0.000} C_DIS
LIN {X -288.697,Y 27.465,Z 125.974,A -5.434,B 90.000,C 0.000} C_DIS
LIN {X -288.707,Y 27.352,Z 128.472,A -5.412,B 90.000,C 0.000} C_DIS
LIN {X -288.709,Y 27.333,Z 130.971,A -5.408,B 90.000,C 0.000} C_DIS
LIN {X -288.713,Y 27.286,Z 133.471,A -5.399,B 90.000,C 0.000} C_DIS
LIN {X -288.722,Y 27.198,Z 135.969,A -5.382,B 90.000,C 0.000} C_DIS
LIN {X -288.722,Y 27.193,Z 138.469,A -5.381,B 90.000,C 0.000} C_DIS
LIN {X -288.722,Y 27.193,Z 139.296,A -5.381,B 90.000,C 0.000} C_DIS
LIN {X -288.848,Y 25.826,Z 139.276,A -5.109,B 90.000,C 0.000} C_DIS
LIN {X -288.883,Y 25.430,Z 139.172,A -5.031,B 90.000,C 0.000} C_DIS
LIN {X -288.964,Y 24.494,Z 139.131,A -4.845,B 90.000,C 0.000} C_DIS
LIN {X -288.996,Y 24.116,Z 139.027,A -4.770,B 90.000,C 0.000} C_DIS
LIN {X -289.081,Y 23.072,Z 138.987,A -4.563,B 90.000,C 0.000} C_DIS
LIN {X -289.111,Y 22.693,Z 138.882,A -4.488,B 90.000,C 0.000} C_DIS
LIN {X -289.183,Y 21.757,Z 138.842,A -4.303,B 90.000,C 0.000} C_DIS
LIN {X -289.210,Y 21.386,Z 138.738,A -4.229,B 90.000,C 0.000} C_DIS
LIN {X -289.283,Y 20.381,Z 138.703,A -4.030,B 90.000,C 0.000} C_DIS
LIN {X -289.302,Y 20.114,Z 138.615,A -3.977,B 90.000,C 0.000} C_DIS
LIN {X -289.306,Y 20.046,Z 138.523,A -3.964,B 90.000,C 0.000} C_DIS
LIN {X -289.309,Y 20.009,Z 138.390,A -3.956,B 90.000,C 0.000} C_DIS
LIN {X -289.310,Y 19.991,Z 137.417,A -3.953,B 90.000,C 0.000} C_DIS
LIN {X -289.344,Y 19.499,Z 137.396,A -3.855,B 90.000,C 0.000} C_DIS
LIN {X -289.349,Y 19.414,Z 137.345,A -3.839,B 90.000,C 0.000} C_DIS
LIN {X -289.359,Y 19.270,Z 137.293,A -3.810,B 90.000,C 0.000} C_DIS
LIN {X -289.406,Y 18.549,Z 137.252,A -3.667,B 90.000,C 0.000} C_DIS
LIN {X -289.426,Y 18.242,Z 137.148,A -3.607,B 90.000,C 0.000} C_DIS
LIN {X -289.477,Y 17.413,Z 137.108,A -3.442,B 90.000,C 0.000} C_DIS
LIN {X -289.496,Y 17.088,Z 137.004,A -3.378,B 90.000,C 0.000} C_DIS
LIN {X -289.544,Y 16.258,Z 136.963,A -3.214,B 90.000,C 0.000} C_DIS
LIN {X -289.561,Y 15.952,Z 136.860,A -3.153,B 90.000,C 0.000} C_DIS
LIN {X -289.600,Y 15.230,Z 136.818,A -3.010,B 90.000,C 0.000} C_DIS
LIN {X -289.615,Y 14.942,Z 136.715,A -2.953,B 90.000,C 0.000} C_DIS
LIN {X -289.654,Y 14.164,Z 136.672,A -2.800,B 90.000,C 0.000} C_DIS
LIN {X -289.657,Y 14.093,Z 136.633,A -2.785,B 90.000,C 0.000} C_DIS
LIN {X -289.660,Y 14.033,Z 136.444,A -2.774,B 90.000,C 0.000} C_DIS
LIN {X -289.670,Y 13.829,Z 136.230,A -2.733,B 90.000,C 0.000} C_DIS
LIN {X -289.675,Y 13.723,Z 136.000,A -2.712,B 90.000,C 0.000} C_DIS
LIN {X -289.746,Y 12.139,Z 134.067,A -2.399,B 90.000,C 0.000} C_DIS
LIN {X -289.755,Y 11.910,Z 133.806,A -2.354,B 90.000,C 0.000} C_DIS
LIN {X -289.760,Y 11.788,Z 133.627,A -2.330,B 90.000,C 0.000} C_DIS
LIN {X -289.783,Y 11.219,Z 133.058,A -2.217,B 90.000,C 0.000} C_DIS
LIN {X -289.790,Y 11.041,Z 132.937,A -2.182,B 90.000,C 0.000} C_DIS
LIN {X -289.857,Y 9.115,Z 131.345,A -1.801,B 90.000,C 0.000} C_DIS
LIN {X -289.865,Y 8.849,Z 131.122,A -1.749,B 90.000,C 0.000} C_DIS
LIN {X -289.872,Y 8.618,Z 131.015,A -1.703,B 90.000,C 0.000} C_DIS
LIN {X -289.878,Y 8.404,Z 130.811,A -1.661,B 90.000,C 0.000} C_DIS
LIN {X -289.882,Y 8.283,Z 130.769,A -1.637,B 90.000,C 0.000} C_DIS
LIN {X -289.884,Y 8.192,Z 130.748,A -1.619,B 90.000,C 0.000} C_DIS
LIN {X -289.886,Y 8.116,Z 130.645,A -1.604,B 90.000,C 0.000} C_DIS
LIN {X -289.889,Y 8.026,Z 130.624,A -1.586,B 90.000,C 0.000} C_DIS
LIN {X -289.892,Y 7.904,Z 130.582,A -1.562,B 90.000,C 0.000} C_DIS
LIN {X -289.898,Y 7.682,Z 130.378,A -1.518,B 90.000,C 0.000} C_DIS
LIN {X -289.901,Y 7.560,Z 130.335,A -1.494,B 90.000,C 0.000} C_DIS
LIN {X -289.904,Y 7.470,Z 130.314,A -1.476,B 90.000,C 0.000} C_DIS
LIN {X -289.906,Y 7.389,Z 130.212,A -1.460,B 90.000,C 0.000} C_DIS
LIN {X -289.911,Y 7.185,Z 130.169,A -1.420,B 90.000,C 0.000} C_DIS
LIN {X -289.913,Y 7.100,Z 130.067,A -1.403,B 90.000,C 0.000} C_DIS
LIN {X -289.918,Y 6.896,Z 130.025,A -1.363,B 90.000,C 0.000} C_DIS
LIN {X -289.920,Y 6.811,Z 129.923,A -1.346,B 90.000,C 0.000} C_DIS
LIN {X -289.925,Y 6.607,Z 129.880,A -1.306,B 90.000,C 0.000} C_DIS
LIN {X -289.927,Y 6.523,Z 129.778,A -1.289,B 90.000,C 0.000} C_DIS
LIN {X -289.931,Y 6.318,Z 129.736,A -1.248,B 90.000,C 0.000} C_DIS
LIN {X -289.933,Y 6.234,Z 129.634,A -1.232,B 90.000,C 0.000} C_DIS
LIN {X -289.937,Y 6.029,Z 129.591,A -1.191,B 90.000,C 0.000} C_DIS
LIN {X -289.938,Y 5.987,Z 129.540,A -1.183,B 90.000,C 0.000} C_DIS
LIN {X -289.940,Y 5.923,Z 129.489,A -1.170,B 90.000,C 0.000} C_DIS
LIN {X -289.946,Y 5.617,Z 129.447,A -1.110,B 90.000,C 0.000} C_DIS
LIN {X -289.947,Y 5.553,Z 129.396,A -1.097,B 90.000,C 0.000} C_DIS
LIN {X -289.948,Y 5.511,Z 129.345,A -1.089,B 90.000,C 0.000} C_DIS
LIN {X -289.951,Y 5.307,Z 129.302,A -1.049,B 90.000,C 0.000} C_DIS
LIN {X -289.952,Y 5.264,Z 129.251,A -1.040,B 90.000,C 0.000} C_DIS
LIN {X -289.953,Y 5.201,Z 129.200,A -1.028,B 90.000,C 0.000} C_DIS
LIN {X -289.959,Y 4.895,Z 129.158,A -0.967,B 90.000,C 0.000} C_DIS
LIN {X -289.961,Y 4.767,Z 129.056,A -0.942,B 90.000,C 0.000} C_DIS
LIN {X -289.966,Y 4.461,Z 129.013,A -0.881,B 90.000,C 0.000} C_DIS
LIN {X -289.968,Y 4.334,Z 128.911,A -0.856,B 90.000,C 0.000} C_DIS
LIN {X -289.972,Y 4.028,Z 128.869,A -0.796,B 90.000,C 0.000} C_DIS
LIN {X -289.973,Y 3.964,Z 128.818,A -0.783,B 90.000,C 0.000} C_DIS
LIN {X -289.974,Y 3.879,Z 128.767,A -0.766,B 90.000,C 0.000} C_DIS
LIN {X -289.979,Y 3.471,Z 128.724,A -0.686,B 90.000,C 0.000} C_DIS
LIN {X -289.981,Y 3.280,Z 128.622,A -0.648,B 90.000,C 0.000} C_DIS
LIN {X -289.987,Y 2.769,Z 128.580,A -0.547,B 90.000,C 0.000} C_DIS
LIN {X -289.989,Y 2.537,Z 128.477,A -0.501,B 90.000,C 0.000} C_DIS
LIN {X -289.994,Y 1.923,Z 128.435,A -0.380,B 90.000,C 0.000} C_DIS
LIN {X -289.994,Y 1.796,Z 128.384,A -0.355,B 90.000,C 0.000} C_DIS
LIN {X -289.996,Y 1.579,Z 128.332,A -0.312,B 90.000,C 0.000} C_DIS
LIN {X -290.000,Y 0.423,Z 128.292,A -0.084,B 90.000,C 0.000} C_DIS
LIN {X -290.000,Y 0.008,Z 128.187,A -0.001,B 90.000,C 0.000} C_DIS
LIN {X -289.998,Y -1.040,Z 128.187,A 0.206,B 90.000,C 0.000} C_DIS
LIN {X -289.996,Y -1.456,Z 128.292,A 0.288,B 90.000,C 0.000} C_DIS
LIN {X -289.988,Y -2.612,Z 128.332,A 0.516,B 90.000,C 0.000} C_DIS
LIN {X -289.986,Y -2.829,Z 128.384,A 0.559,B 90.000,C 0.000} C_DIS
LIN {X -289.985,Y -2.935,Z 128.435,A 0.580,B 90.000,C 0.000} C_DIS
LIN {X -289.980,Y -3.445,Z 128.478,A 0.681,B 90.000,C 0.000} C_DIS
LIN {X -289.977,Y -3.658,Z 128.580,A 0.723,B 90.000,C 0.000} C_DIS
LIN {X -289.970,Y -4.168,Z 128.622,A 0.823,B 90.000,C 0.000} C_DIS
LIN {X -289.969,Y -4.274,Z 128.673,A 0.844,B 90.000,C 0.000} C_DIS
LIN {X -289.968,Y -4.338,Z 128.724,A 0.857,B 90.000,C 0.000} C_DIS
LIN {X -289.963,Y -4.644,Z 128.767,A 0.918,B 90.000,C 0.000} C_DIS
LIN {X -289.962,Y -4.707,Z 128.818,A 0.930,B 90.000,C 0.000} C_DIS
LIN {X -289.960,Y -4.792,Z 128.869,A 0.947,B 90.000,C 0.000} C_DIS
LIN {X -289.953,Y -5.201,Z 128.911,A 1.028,B 90.000,C 0.000} C_DIS
LIN {X -289.952,Y -5.286,Z 128.962,A 1.044,B 90.000,C 0.000} C_DIS
LIN {X -289.951,Y -5.349,Z 129.013,A 1.057,B 90.000,C 0.000} C_DIS
LIN {X -289.945,Y -5.655,Z 129.056,A 1.117,B 90.000,C 0.000} C_DIS
LIN {X -289.944,Y -5.719,Z 129.107,A 1.130,B 90.000,C 0.000} C_DIS
LIN {X -289.943,Y -5.761,Z 129.158,A 1.138,B 90.000,C 0.000} C_DIS
LIN {X -289.939,Y -5.966,Z 129.200,A 1.179,B 90.000,C 0.000} C_DIS
LIN {X -289.938,Y -6.008,Z 129.251,A 1.187,B 90.000,C 0.000} C_DIS
LIN {X -289.936,Y -6.072,Z 129.302,A 1.200,B 90.000,C 0.000} C_DIS
LIN {X -289.930,Y -6.378,Z 129.345,A 1.260,B 90.000,C 0.000} C_DIS
LIN {X -289.928,Y -6.442,Z 129.396,A 1.273,B 90.000,C 0.000} C_DIS
LIN {X -289.928,Y -6.484,Z 129.447,A 1.281,B 90.000,C 0.000} C_DIS
LIN {X -289.923,Y -6.688,Z 129.489,A 1.321,B 90.000,C 0.000} C_DIS
LIN {X -289.921,Y -6.773,Z 129.591,A 1.338,B 90.000,C 0.000} C_DIS
LIN {X -289.916,Y -6.977,Z 129.634,A 1.379,B 90.000,C 0.000} C_DIS
LIN {X -289.914,Y -7.062,Z 129.736,A 1.395,B 90.000,C 0.000} C_DIS
LIN {X -289.909,Y -7.266,Z 129.778,A 1.436,B 90.000,C 0.000} C_DIS
LIN {X -289.907,Y -7.351,Z 129.880,A 1.452,B 90.000,C 0.000} C_DIS
LIN {X -289.902,Y -7.555,Z 129.923,A 1.493,B 90.000,C 0.000} C_DIS
LIN {X -289.899,Y -7.640,Z 130.025,A 1.510,B 90.000,C 0.000} C_DIS
LIN {X -289.894,Y -7.844,Z 130.067,A 1.550,B 90.000,C 0.000} C_DIS
LIN {X -289.892,Y -7.924,Z 130.169,A 1.566,B 90.000,C 0.000} C_DIS
LIN {X -289.889,Y -8.015,Z 130.191,A 1.584,B 90.000,C 0.000} C_DIS
LIN {X -289.886,Y -8.136,Z 130.233,A 1.608,B 90.000,C 0.000} C_DIS
LIN {X -289.880,Y -8.354,Z 130.437,A 1.651,B 90.000,C 0.000} C_DIS
LIN {X -289.873,Y -8.574,Z 130.522,A 1.694,B 90.000,C 0.000} C_DIS
LIN {X -289.867,Y -8.788,Z 130.726,A 1.736,B 90.000,C 0.000} C_DIS
LIN {X -289.860,Y -9.008,Z 130.811,A 1.780,B 90.000,C 0.000} C_DIS
LIN {X -289.853,Y -9.217,Z 131.015,A 1.821,B 90.000,C 0.000} C_DIS
LIN {X -289.846,Y -9.448,Z 131.122,A 1.867,B 90.000,C 0.000} C_DIS
LIN {X -289.780,Y -11.293,Z 132.806,A 2.232,B 90.000,C 0.000} C_DIS
LIN {X -289.709,Y -12.977,Z 134.653,A 2.565,B 90.000,C 0.000} C_DIS
LIN {X -289.708,Y -13.001,Z 134.679,A 2.570,B 90.000,C 0.000} C_DIS
LIN {X -289.705,Y -13.086,Z 134.830,A 2.586,B 90.000,C 0.000} C_DIS
LIN {X -289.698,Y -13.230,Z 135.032,A 2.615,B 90.000,C 0.000} C_DIS
LIN {X -289.693,Y -13.332,Z 135.139,A 2.635,B 90.000,C 0.000} C_DIS
LIN {X -289.689,Y -13.417,Z 135.359,A 2.652,B 90.000,C 0.000} C_DIS
LIN {X -289.680,Y -13.621,Z 135.573,A 2.692,B 90.000,C 0.000} C_DIS
LIN {X -289.676,Y -13.706,Z 135.793,A 2.709,B 90.000,C 0.000} C_DIS
LIN {X -289.666,Y -13.910,Z 136.011,A 2.749,B 90.000,C 0.000} C_DIS
LIN {X -289.664,Y -13.952,Z 136.132,A 2.758,B 90.000,C 0.000} C_DIS
LIN {X -289.663,Y -13.973,Z 136.223,A 2.762,B 90.000,C 0.000} C_DIS
LIN {X -289.658,Y -14.075,Z 136.294,A 2.782,B 90.000,C 0.000} C_DIS
LIN {X -289.655,Y -14.134,Z 136.521,A 2.794,B 90.000,C 0.000} C_DIS
LIN {X -289.649,Y -14.254,Z 136.620,A 2.817,B 90.000,C 0.000} C_DIS
LIN {X -289.639,Y -14.465,Z 136.677,A 2.859,B 90.000,C 0.000} C_DIS
LIN {X -289.606,Y -15.115,Z 136.715,A 2.988,B 90.000,C 0.000} C_DIS
LIN {X -289.591,Y -15.396,Z 136.818,A 3.043,B 90.000,C 0.000} C_DIS
LIN {X -289.552,Y -16.117,Z 136.860,A 3.186,B 90.000,C 0.000} C_DIS
LIN {X -289.535,Y -16.424,Z 136.963,A 3.247,B 90.000,C 0.000} C_DIS
LIN {X -289.486,Y -17.253,Z 137.004,A 3.411,B 90.000,C 0.000} C_DIS
LIN {X -289.467,Y -17.578,Z 137.108,A 3.475,B 90.000,C 0.000} C_DIS
LIN {X -289.415,Y -18.407,Z 137.148,A 3.639,B 90.000,C 0.000} C_DIS
LIN {X -289.394,Y -18.732,Z 137.252,A 3.703,B 90.000,C 0.000} C_DIS
LIN {X -289.340,Y -19.561,Z 137.293,A 3.868,B 90.000,C 0.000} C_DIS
LIN {X -289.329,Y -19.723,Z 137.345,A 3.900,B 90.000,C 0.000} C_DIS
LIN {X -289.324,Y -19.787,Z 137.396,A 3.912,B 90.000,C 0.000} C_DIS
LIN {X -289.314,Y -19.940,Z 137.417,A 3.943,B 90.000,C 0.000} C_DIS
LIN {X -289.299,Y -20.156,Z 137.417,A 3.985,B 90.000,C 0.000} C_DIS
LIN {X -289.297,Y -20.174,Z 138.386,A 3.989,B 90.000,C 0.000} C_DIS
LIN {X -289.291,Y -20.273,Z 138.611,A 4.009,B 90.000,C 0.000} C_DIS
LIN {X -289.273,Y -20.519,Z 138.701,A 4.057,B 90.000,C 0.000} C_DIS
LIN {X -289.207,Y -21.425,Z 138.738,A 4.237,B 90.000,C 0.000} C_DIS
LIN {X -289.180,Y -21.795,Z 138.843,A 4.310,B 90.000,C 0.000} C_DIS
LIN {X -289.099,Y -22.840,Z 138.882,A 4.517,B 90.000,C 0.000} C_DIS
LIN {X -289.066,Y -23.254,Z 138.987,A 4.599,B 90.000,C 0.000} C_DIS
LIN {X -288.971,Y -24.407,Z 139.027,A 4.828,B 90.000,C 0.000} C_DIS
LIN {X -288.936,Y -24.821,Z 139.132,A 4.910,B 90.000,C 0.000} C_DIS
LIN {X -288.844,Y -25.865,Z 139.171,A 5.117,B 90.000,C 0.000} C_DIS
LIN {X -288.813,Y -26.206,Z 139.275,A 5.185,B 90.000,C 0.000} C_DIS
LIN {X -288.734,Y -27.070,Z 139.296,A 5.356,B 90.000,C 0.000} C_DIS
LIN {X -288.734,Y -27.070,Z 136.796,A 5.356,B 90.000,C 0.000} C_DIS
LIN {X -288.731,Y -27.105,Z 134.296,A 5.363,B 90.000,C 0.000} C_DIS
LIN {X -288.721,Y -27.204,Z 131.799,A 5.383,B 90.000,C 0.000} C_DIS
LIN {X -288.719,Y -27.223,Z 129.299,A 5.386,B 90.000,C 0.000} C_DIS
LIN {X -288.711,Y -27.308,Z 126.800,A 5.403,B 90.000,C 0.000} C_DIS
LIN {X -288.707,Y -27.354,Z 124.301,A 5.412,B 90.000,C 0.000} C_DIS
LIN {X -288.705,Y -27.373,Z 121.801,A 5.416,B 90.000,C 0.000} C_DIS
LIN {X -288.695,Y -27.486,Z 119.304,A 5.439,B 90.000,C 0.000} C_DIS
LIN {X -288.693,Y -27.504,Z 116.804,A 5.442,B 90.000,C 0.000} C_DIS
LIN {X -288.690,Y -27.537,Z 114.304,A 5.449,B 90.000,C 0.000} C_DIS
LIN {X -288.686,Y -27.574,Z 113.714,A 5.456,B 90.000,C 0.000} C_DIS
LIN {X -288.681,Y -27.625,Z 113.651,A 5.466,B 90.000,C 0.000} C_DIS
LIN {X -288.679,Y -27.646,Z 113.498,A 5.470,B 90.000,C 0.000} C_DIS
LIN {X -288.681,Y -27.625,Z 113.344,A 5.466,B 90.000,C 0.000} C_DIS
LIN {X -288.686,Y -27.574,Z 113.281,A 5.456,B 90.000,C 0.000} C_DIS
LIN {X -288.691,Y -27.523,Z 113.175,A 5.446,B 90.000,C 0.000} C_DIS
LIN {X -288.695,Y -27.481,Z 112.664,A 5.438,B 90.000,C 0.000} C_DIS
LIN {X -288.705,Y -27.379,Z 112.452,A 5.417,B 90.000,C 0.000} C_DIS
LIN {X -288.709,Y -27.337,Z 111.942,A 5.409,B 90.000,C 0.000} C_DIS
LIN {X -288.718,Y -27.235,Z 111.751,A 5.389,B 90.000,C 0.000} C_DIS
LIN {X -288.722,Y -27.193,Z 111.342,A 5.380,B 90.000,C 0.000} C_DIS
LIN {X -288.732,Y -27.091,Z 111.172,A 5.360,B 90.000,C 0.000} C_DIS
LIN {X -288.736,Y -27.049,Z 110.764,A 5.352,B 90.000,C 0.000} C_DIS
LIN {X -288.745,Y -26.947,Z 110.573,A 5.332,B 90.000,C 0.000} C_DIS
LIN {X -288.749,Y -26.905,Z 110.063,A 5.323,B 90.000,C 0.000} C_DIS
LIN {X -288.759,Y -26.803,Z 109.872,A 5.303,B 90.000,C 0.000} C_DIS
LIN {X -288.763,Y -26.761,Z 109.463,A 5.295,B 90.000,C 0.000} C_DIS
LIN {X -288.772,Y -26.660,Z 109.272,A 5.275,B 90.000,C 0.000} C_DIS
LIN {X -288.776,Y -26.617,Z 108.762,A 5.266,B 90.000,C 0.000} C_DIS
LIN {X -288.785,Y -26.516,Z 108.571,A 5.246,B 90.000,C 0.000} C_DIS
LIN {X -288.789,Y -26.473,Z 108.163,A 5.238,B 90.000,C 0.000} C_DIS
LIN {X -288.798,Y -26.372,Z 107.993,A 5.218,B 90.000,C 0.000} C_DIS
LIN {X -288.802,Y -26.329,Z 107.585,A 5.209,B 90.000,C 0.000} C_DIS
LIN {X -288.812,Y -26.228,Z 107.394,A 5.189,B 90.000,C 0.000} C_DIS
LIN {X -288.815,Y -26.185,Z 106.883,A 5.181,B 90.000,C 0.000} C_DIS
LIN {X -288.825,Y -26.084,Z 106.692,A 5.160,B 90.000,C 0.000} C_DIS
LIN {X -288.828,Y -26.042,Z 106.284,A 5.152,B 90.000,C 0.000} C_DIS
LIN {X -288.838,Y -25.940,Z 106.114,A 5.132,B 90.000,C 0.000} C_DIS
LIN {X -288.841,Y -25.898,Z 105.706,A 5.123,B 90.000,C 0.000} C_DIS
LIN {X -288.850,Y -25.796,Z 105.525,A 5.103,B 90.000,C 0.000} C_DIS
LIN {X -288.852,Y -25.775,Z 105.293,A 5.099,B 90.000,C 0.000} C_DIS
LIN {X -288.848,Y -25.820,Z 104.980,A 5.108,B 90.000,C 0.000} C_DIS
LIN {X -288.830,Y -26.024,Z 104.715,A 5.149,B 90.000,C 0.000} C_DIS
LIN {X -288.811,Y -26.233,Z 104.538,A 5.190,B 90.000,C 0.000} C_DIS
LIN {X -288.797,Y -26.384,Z 104.465,A 5.220,B 90.000,C 0.000} C_DIS
LIN {X -288.790,Y -26.462,Z 104.443,A 5.235,B 90.000,C 0.000} C_DIS
LIN {X -288.787,Y -26.494,Z 104.392,A 5.242,B 90.000,C 0.000} C_DIS
LIN {X -288.771,Y -26.674,Z 104.340,A 5.278,B 90.000,C 0.000} C_DIS
LIN {X -288.665,Y -27.789,Z 104.320,A 5.499,B 90.000,C 0.000} C_DIS
LIN {X -288.664,Y -27.809,Z 102.315,A 5.503,B 90.000,C 0.000} C_DIS
LIN {X -288.659,Y -27.861,Z 102.008,A 5.513,B 90.000,C 0.000} C_DIS
LIN {X -288.654,Y -27.912,Z 101.970,A 5.523,B 90.000,C 0.000} C_DIS
LIN {X -288.652,Y -27.933,Z 101.879,A 5.527,B 90.000,C 0.000} C_DIS
LIN {X -288.647,Y -27.976,Z 101.758,A 5.536,B 90.000,C 0.000} C_DIS
LIN {X -288.638,Y -28.077,Z 101.646,A 5.556,B 90.000,C 0.000} C_DIS
LIN {X -288.611,Y -28.348,Z 101.253,A 5.610,B 90.000,C 0.000} C_DIS
LIN {X -288.446,Y -29.979,Z 99.366,A 5.934,B 90.000,C 0.000} C_DIS
LIN {X -288.275,Y -31.586,Z 97.458,A 6.253,B 90.000,C 0.000} C_DIS
LIN {X -288.093,Y -33.203,Z 95.560,A 6.574,B 90.000,C 0.000} C_DIS
LIN {X -287.902,Y -34.819,Z 93.662,A 6.896,B 90.000,C 0.000} C_DIS
LIN {X -287.703,Y -36.424,Z 91.756,A 7.215,B 90.000,C 0.000} C_DIS
LIN {X -287.495,Y -38.035,Z 89.856,A 7.536,B 90.000,C 0.000} C_DIS
LIN {X -287.277,Y -39.647,Z 87.958,A 7.858,B 90.000,C 0.000} C_DIS
LIN {X -287.050,Y -41.258,Z 86.060,A 8.179,B 90.000,C 0.000} C_DIS
